LIN {X 0,Y 457.306,Z 988.134,A -85,B 0,C 180,E1 20807.433,E2 20807.433} C_VEL
LIN {X 0,Y 456.621,Z 997.32,A -85,B 0,C 180,E1 20804.572,E2 20804.572} C_VEL
LIN {X 0,Y 456.252,Z 1003.948,A -85,B 0,C 180,E1 20802.019,E2 20802.019} C_VEL
LIN {X 0,Y 456.036,Z 1009.804,A -85,B 0,C 180,E1 20799.213,E2 20799.213} C_VEL
LIN {X 0,Y 455.944,Z 1013.955,A -85,B 0,C 180,E1 20796.424,E2 20796.424} C_VEL
LIN {X 0,Y 455.898,Z 1016.711,A -85,B 0,C 180,E1 20793.65,E2 20793.65} C_VEL
LIN {X 0,Y 455.893,Z 1017.826,A -85,B 0,C 180,E1 20791.009,E2 20791.009} C_VEL
LIN {X 0,Y 455.907,Z 1017.736,A -85,B 0,C 180,E1 20788.495,E2 20788.495} C_VEL
LIN {X 0,Y 455.909,Z 1016.072,A -85,B 0,C 180,E1 20785.601,E2 20785.601} C_VEL
LIN {X 0,Y 455.929,Z 1013.324,A -85,B 0,C 180,E1 20783.076,E2 20783.076} C_VEL
LIN {X 0,Y 456.046,Z 1008.598,A -85,B 0,C 180,E1 20780.157,E2 20780.157} C_VEL
LIN {X 0,Y 456.297,Z 1003.054,A -85,B 0,C 180,E1 20777.603,E2 20777.603} C_VEL
LIN {X 0,Y 456.792,Z 994.97,A -85,B 0,C 180,E1 20774.646,E2 20774.646} C_VEL
LIN {X 0,Y 457.47,Z 986.327,A -85,B 0,C 180,E1 20772.055,E2 20772.055} C_VEL
LIN {X 0,Y 458.57,Z 974.884,A -85,B 0,C 180,E1 20769.186,E2 20769.186} C_VEL
LIN {X 0,Y 460.023,Z 962.425,A -85,B 0,C 180,E1 20766.521,E2 20766.521} C_VEL
LIN {X 0,Y 461.835,Z 948.135,A -85,B 0,C 180,E1 20763.933,E2 20763.933} C_VEL
LIN {X 0,Y 464.103,Z 931.673,A -85,B 0,C 180,E1 20761.362,E2 20761.362} C_VEL
LIN {X 0,Y 466.448,Z 915.582,A -85,B 0,C 180,E1 20759.187,E2 20759.187} C_VEL
LIN {X 0,Y 468.956,Z 897.768,A -85,B 0,C 180,E1 20757.144,E2 20757.144} C_VEL
LIN {X 0,Y 471.66,Z 878.612,A -85,B 0,C 180,E1 20755.238,E2 20755.238} C_VEL
LIN {X 0,Y 474.23,Z 859.23,A -85,B 0,C 180,E1 20753.599,E2 20753.599} C_VEL
LIN {X 0,Y 476.999,Z 837.541,A -85,B 0,C 180,E1 20752.038,E2 20752.038} C_VEL
LIN {X 0,Y 479.213,Z 818.309,A -85,B 0,C 180,E1 20750.878,E2 20750.878} C_VEL
LIN {X 0,Y 481.581,Z 794.779,A -85,B 0,C 180,E1 20749.71,E2 20749.71} C_VEL
LIN {X 0,Y 483.484,Z 773.134,A -85,B 0,C 180,E1 20748.864,E2 20748.864} C_VEL
LIN {X 0,Y 485.004,Z 750.7,A -85,B 0,C 180,E1 20748.207,E2 20748.207} C_VEL
LIN {X 0,Y 486.043,Z 728.316,A -85,B 0,C 180,E1 20747.734,E2 20747.734} C_VEL
LIN {X 0,Y 491.395,Z 520.554,A -85,B 0,C 180,E1 20744.158,E2 20744.158} C_VEL
LIN {X 0,Y 493.752,Z 431.767,A -85,B 0,C 180,E1 20742.581,E2 20742.581} C_VEL
LIN {X 0,Y 480.639,Z 411.465,A -85,B 0,C 180,E1 20740.421,E2 20740.421} C_VEL
LIN {X 0,Y 467.607,Z 392.801,A -85,B 0,C 180,E1 20738.088,E2 20738.088} C_VEL
LIN {X 0,Y 463.585,Z 387.256,A -85,B 0,C 180,E1 20737.305,E2 20737.305} C_VEL
LIN {X 0,Y 458.876,Z 378.323,A -85,B 0,C 180,E1 20735.575,E2 20735.575} C_VEL
LIN {X 0,Y 457.213,Z 375.183,A -85,B 0,C 180,E1 20734.917,E2 20734.917} C_VEL
LIN {X 0,Y 457.035,Z 374.27,A -85,B 0,C 180,E1 20734.665,E2 20734.665} C_VEL
LIN {X 0,Y 456.993,Z 374.085,A -85,B 0,C 180,E1 20731.087,E2 20731.087} C_VEL
LIN {X 0,Y 457.016,Z 374.122,A -85,B 0,C 180,E1 20727.492,E2 20727.492} C_VEL
LIN {X 0,Y 457.052,Z 374.11,A -85,B 0,C 180,E1 20723.873,E2 20723.873} C_VEL
LIN {X 0,Y 457.006,Z 374.114,A -85,B 0,C 180,E1 20720.356,E2 20720.356} C_VEL
LIN {X 0,Y 457,Z 374.117,A -85,B 0,C 180,E1 20716.655,E2 20716.655} C_VEL
LIN {X 0,Y 457.035,Z 374.118,A -85,B 0,C 180,E1 20713.151,E2 20713.151} C_VEL
LIN {X 0,Y 457.061,Z 374.117,A -85,B 0,C 180,E1 20709.443,E2 20709.443} C_VEL
LIN {X 0,Y 457.02,Z 374.12,A -85,B 0,C 180,E1 20705.901,E2 20705.901} C_VEL
LIN {X 0,Y 457.012,Z 374.117,A -85,B 0,C 180,E1 20702.257,E2 20702.257} C_VEL
LIN {X 0,Y 457.045,Z 374.111,A -85,B 0,C 180,E1 20698.746,E2 20698.746} C_VEL
LIN {X 0,Y 457.066,Z 374.108,A -85,B 0,C 180,E1 20695.105,E2 20695.105} C_VEL
LIN {X 0,Y 457.027,Z 374.117,A -85,B 0,C 180,E1 20691.571,E2 20691.571} C_VEL
LIN {X 0,Y 457.024,Z 374.114,A -85,B 0,C 180,E1 20687.876,E2 20687.876} C_VEL
LIN {X 0,Y 457.051,Z 374.108,A -85,B 0,C 180,E1 20684.252,E2 20684.252} C_VEL
LIN {X 0,Y 457.075,Z 374.104,A -85,B 0,C 180,E1 20680.579,E2 20680.579} C_VEL
LIN {X 0,Y 457.049,Z 374.11,A -85,B 0,C 180,E1 20676.946,E2 20676.946} C_VEL
LIN {X 0,Y 457.034,Z 374.112,A -85,B 0,C 180,E1 20673.353,E2 20673.353} C_VEL
LIN {X 0,Y 457.054,Z 374.105,A -85,B 0,C 180,E1 20669.771,E2 20669.771} C_VEL
LIN {X 0,Y 457.078,Z 374.103,A -85,B 0,C 180,E1 20666.095,E2 20666.095} C_VEL
LIN {X 0,Y 457.069,Z 374.106,A -85,B 0,C 180,E1 20662.355,E2 20662.355} C_VEL
LIN {X 0,Y 457.044,Z 374.106,A -85,B 0,C 180,E1 20658.805,E2 20658.805} C_VEL
LIN {X 0,Y 457.05,Z 374.113,A -85,B 0,C 180,E1 20655.04,E2 20655.04} C_VEL
LIN {X 0,Y 457.075,Z 374.112,A -85,B 0,C 180,E1 20651.342,E2 20651.342} C_VEL
LIN {X 0,Y 457.073,Z 374.105,A -85,B 0,C 180,E1 20647.607,E2 20647.607} C_VEL
LIN {X 0,Y 457.074,Z 374.108,A -85,B 0,C 180,E1 20643.9,E2 20643.9} C_VEL
LIN {X 0,Y 457.051,Z 374.08,A -85,B 0,C 180,E1 20640.204,E2 20640.204} C_VEL
LIN {X 0,Y 457.056,Z 374.087,A -85,B 0,C 180,E1 20636.5,E2 20636.5} C_VEL
LIN {X 0,Y 457.075,Z 374.098,A -85,B 0,C 180,E1 20632.775,E2 20632.775} C_VEL
LIN {X 0,Y 457.119,Z 374.398,A -85,B 0,C 180,E1 20631.555,E2 20631.555} C_VEL
LIN {X 0,Y 457.57,Z 376.045,A -85,B 0,C 180,E1 20631.29,E2 20631.29} C_VEL
LIN {X 0,Y 459.613,Z 379.002,A -85,B 0,C 180,E1 20630.876,E2 20630.876} C_VEL
LIN {X 0,Y 461.397,Z 380.643,A -85,B 0,C 180,E1 20630.548,E2 20630.548} C_VEL
LIN {X 0,Y 463.85,Z 384.388,A -85,B 0,C 180,E1 20630.067,E2 20630.067} C_VEL
LIN {X 0,Y 465.76,Z 386.443,A -85,B 0,C 180,E1 20629.721,E2 20629.721} C_VEL
LIN {X 0,Y 469.06,Z 390.773,A -85,B 0,C 180,E1 20629.118,E2 20629.118} C_VEL
LIN {X 0,Y 469.173,Z 390.881,A -85,B 0,C 180,E1 20629.098,E2 20629.098} C_VEL
LIN {X 0,Y 470.97,Z 393.832,A -85,B 0,C 180,E1 20628.762,E2 20628.762} C_VEL
LIN {X 0,Y 472.42,Z 399.823,A -85,B 0,C 180,E1 20628.407,E2 20628.407} C_VEL
LIN {X 0,Y 473.933,Z 407.518,A -85,B 0,C 180,E1 20628.004,E2 20628.004} C_VEL
LIN {X 0,Y 475.539,Z 410.916,A -85,B 0,C 180,E1 20627.694,E2 20627.694} C_VEL
LIN {X 0,Y 486.708,Z 426.723,A -85,B 0,C 180,E1 20625.82,E2 20625.82} C_VEL
LIN {X 0,Y 488.009,Z 429.058,A -85,B 0,C 180,E1 20625.601,E2 20625.601} C_VEL
LIN {X 0,Y 481.886,Z 639.66,A -85,B 0,C 180,E1 20621.903,E2 20621.903} C_VEL
LIN {X 0,Y 479.731,Z 713.742,A -85,B 0,C 180,E1 20620.595,E2 20620.595} C_VEL
LIN {X 0,Y 478.332,Z 735.919,A -85,B 0,C 180,E1 20620.01,E2 20620.01} C_VEL
LIN {X 0,Y 476.579,Z 758.024,A -85,B 0,C 180,E1 20619.232,E2 20619.232} C_VEL
LIN {X 0,Y 474.343,Z 779.679,A -85,B 0,C 180,E1 20618.237,E2 20618.237} C_VEL
LIN {X 0,Y 471.889,Z 800.765,A -85,B 0,C 180,E1 20617.056,E2 20617.056} C_VEL
LIN {X 0,Y 469.117,Z 821.678,A -85,B 0,C 180,E1 20615.623,E2 20615.623} C_VEL
LIN {X 0,Y 466.118,Z 842.401,A -85,B 0,C 180,E1 20613.933,E2 20613.933} C_VEL
LIN {X 0,Y 463.189,Z 861.498,A -85,B 0,C 180,E1 20612.1,E2 20612.1} C_VEL
LIN {X 0,Y 460.249,Z 880.136,A -85,B 0,C 180,E1 20609.997,E2 20609.997} C_VEL
LIN {X 0,Y 457.509,Z 897.277,A -85,B 0,C 180,E1 20607.742,E2 20607.742} C_VEL
LIN {X 0,Y 454.98,Z 913.876,A -85,B 0,C 180,E1 20605.207,E2 20605.207} C_VEL
LIN {X 0,Y 452.94,Z 928.382,A -85,B 0,C 180,E1 20602.641,E2 20602.641} C_VEL
LIN {X 0,Y 451.242,Z 941.581,A -85,B 0,C 180,E1 20599.916,E2 20599.916} C_VEL
LIN {X 0,Y 449.92,Z 953.436,A -85,B 0,C 180,E1 20597.026,E2 20597.026} C_VEL
LIN {X 0,Y 448.998,Z 963.452,A -85,B 0,C 180,E1 20594.1,E2 20594.1} C_VEL
LIN {X 0,Y 448.435,Z 971.383,A -85,B 0,C 180,E1 20591.269,E2 20591.269} C_VEL
LIN {X 0,Y 448.117,Z 977.788,A -85,B 0,C 180,E1 20588.395,E2 20588.395} C_VEL
LIN {X 0,Y 447.972,Z 982.717,A -85,B 0,C 180,E1 20585.469,E2 20585.469} C_VEL
LIN {X 0,Y 447.896,Z 985.964,A -85,B 0,C 180,E1 20582.619,E2 20582.619} C_VEL
LIN {X 0,Y 447.884,Z 987.645,A -85,B 0,C 180,E1 20579.846,E2 20579.846} C_VEL
LIN {X 0,Y 447.902,Z 987.873,A -85,B 0,C 180,E1 20577.072,E2 20577.072} C_VEL
LIN {X 0,Y 447.911,Z 986.601,A -85,B 0,C 180,E1 20574.127,E2 20574.127} C_VEL
LIN {X 0,Y 447.948,Z 983.891,A -85,B 0,C 180,E1 20571.316,E2 20571.316} C_VEL
LIN {X 0,Y 448.068,Z 979.465,A -85,B 0,C 180,E1 20568.379,E2 20568.379} C_VEL
LIN {X 0,Y 448.305,Z 973.564,A -85,B 0,C 180,E1 20565.537,E2 20565.537} C_VEL
LIN {X 0,Y 448.786,Z 966.02,A -85,B 0,C 180,E1 20562.672,E2 20562.672} C_VEL
LIN {X 0,Y 449.558,Z 956.85,A -85,B 0,C 180,E1 20559.832,E2 20559.832} C_VEL
LIN {X 0,Y 450.704,Z 945.891,A -85,B 0,C 180,E1 20556.997,E2 20556.997} C_VEL
LIN {X 0,Y 452.212,Z 933.708,A -85,B 0,C 180,E1 20554.32,E2 20554.32} C_VEL
LIN {X 0,Y 454.155,Z 919.628,A -85,B 0,C 180,E1 20551.673,E2 20551.673} C_VEL
LIN {X 0,Y 456.535,Z 903.606,A -85,B 0,C 180,E1 20549.088,E2 20549.088} C_VEL
LIN {X 0,Y 459.226,Z 886.698,A -85,B 0,C 180,E1 20546.726,E2 20546.726} C_VEL
LIN {X 0,Y 462.143,Z 868.394,A -85,B 0,C 180,E1 20544.545,E2 20544.545} C_VEL
LIN {X 0,Y 465.06,Z 849.746,A -85,B 0,C 180,E1 20542.634,E2 20542.634} C_VEL
LIN {X 0,Y 467.9,Z 830.401,A -85,B 0,C 180,E1 20540.957,E2 20540.957} C_VEL
LIN {X 0,Y 470.853,Z 808.986,A -85,B 0,C 180,E1 20539.388,E2 20539.388} C_VEL
LIN {X 0,Y 473.194,Z 790.015,A -85,B 0,C 180,E1 20538.224,E2 20538.224} C_VEL
LIN {X 0,Y 475.597,Z 767.361,A -85,B 0,C 180,E1 20537.083,E2 20537.083} C_VEL
LIN {X 0,Y 477.597,Z 745.324,A -85,B 0,C 180,E1 20536.206,E2 20536.206} C_VEL
LIN {X 0,Y 479.103,Z 723.137,A -85,B 0,C 180,E1 20535.552,E2 20535.552} C_VEL
LIN {X 0,Y 480.178,Z 699.844,A -85,B 0,C 180,E1 20535.06,E2 20535.06} C_VEL
LIN {X 0,Y 485.98,Z 497.309,A -85,B 0,C 180,E1 20531.514,E2 20531.514} C_VEL
LIN {X 0,Y 488.115,Z 428.611,A -85,B 0,C 180,E1 20530.266,E2 20530.266} C_VEL
LIN {X 0,Y 476.772,Z 412.129,A -85,B 0,C 180,E1 20528.29,E2 20528.29} C_VEL
LIN {X 0,Y 469.203,Z 401.84,A -85,B 0,C 180,E1 20526.854,E2 20526.854} C_VEL
LIN {X 0,Y 465.608,Z 397.083,A -85,B 0,C 180,E1 20526.132,E2 20526.132} C_VEL
LIN {X 0,Y 461.979,Z 392.324,A -85,B 0,C 180,E1 20525.38,E2 20525.38} C_VEL
LIN {X 0,Y 458.836,Z 388.242,A -85,B 0,C 180,E1 20524.688,E2 20524.688} C_VEL
LIN {X 0,Y 457.761,Z 386.899,A -85,B 0,C 180,E1 20524.448,E2 20524.448} C_VEL
LIN {X 0,Y 454.797,Z 383.552,A -85,B 0,C 180,E1 20523.782,E2 20523.782} C_VEL
LIN {X 0,Y 453.604,Z 381.346,A -85,B 0,C 180,E1 20523.482,E2 20523.482} C_VEL
LIN {X 0,Y 450.664,Z 378.906,A -85,B 0,C 180,E1 20522.798,E2 20522.798} C_VEL
LIN {X 0,Y 449.291,Z 375.976,A -85,B 0,C 180,E1 20522.366,E2 20522.366} C_VEL
LIN {X 0,Y 449.128,Z 375.128,A -85,B 0,C 180,E1 20521.914,E2 20521.914} C_VEL
LIN {X 0,Y 449.132,Z 375.098,A -85,B 0,C 180,E1 20518.214,E2 20518.214} C_VEL
LIN {X 0,Y 449.135,Z 375.095,A -85,B 0,C 180,E1 20514.507,E2 20514.507} C_VEL
LIN {X 0,Y 449.128,Z 375.103,A -85,B 0,C 180,E1 20510.777,E2 20510.777} C_VEL
LIN {X 0,Y 449.104,Z 375.107,A -85,B 0,C 180,E1 20507.137,E2 20507.137} C_VEL
LIN {X 0,Y 449.103,Z 375.106,A -85,B 0,C 180,E1 20503.443,E2 20503.443} C_VEL
LIN {X 0,Y 449.125,Z 375.104,A -85,B 0,C 180,E1 20499.815,E2 20499.815} C_VEL
LIN {X 0,Y 449.129,Z 375.095,A -85,B 0,C 180,E1 20496.206,E2 20496.206} C_VEL
LIN {X 0,Y 449.092,Z 375.106,A -85,B 0,C 180,E1 20492.558,E2 20492.558} C_VEL
LIN {X 0,Y 449.073,Z 375.108,A -85,B 0,C 180,E1 20488.9,E2 20488.9} C_VEL
LIN {X 0,Y 449.116,Z 375.414,A -85,B 0,C 180,E1 20487.022,E2 20487.022} C_VEL
LIN {X 0,Y 450.636,Z 378.913,A -85,B 0,C 180,E1 20486.158,E2 20486.158} C_VEL
LIN {X 0,Y 451.942,Z 380.731,A -85,B 0,C 180,E1 20485.657,E2 20485.657} C_VEL
LIN {X 0,Y 453.93,Z 384.473,A -85,B 0,C 180,E1 20484.831,E2 20484.831} C_VEL
LIN {X 0,Y 459.557,Z 392.132,A -85,B 0,C 180,E1 20483.523,E2 20483.523} C_VEL
LIN {X 0,Y 466.249,Z 401.457,A -85,B 0,C 180,E1 20482.101,E2 20482.101} C_VEL
LIN {X 0,Y 474.956,Z 414.182,A -85,B 0,C 180,E1 20480.396,E2 20480.396} C_VEL
LIN {X 0,Y 485.83,Z 431.636,A -85,B 0,C 180,E1 20478.436,E2 20478.436} C_VEL
LIN {X 0,Y 488.286,Z 435.985,A -85,B 0,C 180,E1 20478.011,E2 20478.011} C_VEL
LIN {X 0,Y 482.252,Z 637.01,A -85,B 0,C 180,E1 20474.448,E2 20474.448} C_VEL
LIN {X 0,Y 479.387,Z 739.278,A -85,B 0,C 180,E1 20472.658,E2 20472.658} C_VEL
LIN {X 0,Y 477.889,Z 762.53,A -85,B 0,C 180,E1 20472.062,E2 20472.062} C_VEL
LIN {X 0,Y 476.13,Z 784.668,A -85,B 0,C 180,E1 20471.296,E2 20471.296} C_VEL
LIN {X 0,Y 473.953,Z 806.141,A -85,B 0,C 180,E1 20470.328,E2 20470.328} C_VEL
LIN {X 0,Y 471.59,Z 827.058,A -85,B 0,C 180,E1 20469.187,E2 20469.187} C_VEL
LIN {X 0,Y 468.918,Z 847.716,A -85,B 0,C 180,E1 20467.811,E2 20467.811} C_VEL
LIN {X 0,Y 466.071,Z 868.762,A -85,B 0,C 180,E1 20466.156,E2 20466.156} C_VEL
LIN {X 0,Y 463.451,Z 886.719,A -85,B 0,C 180,E1 20464.5,E2 20464.5} C_VEL
LIN {X 0,Y 460.512,Z 906.579,A -85,B 0,C 180,E1 20462.373,E2 20462.373} C_VEL
LIN {X 0,Y 458.095,Z 922.885,A -85,B 0,C 180,E1 20460.353,E2 20460.353} C_VEL
LIN {X 0,Y 455.797,Z 938.318,A -85,B 0,C 180,E1 20458.135,E2 20458.135} C_VEL
LIN {X 0,Y 453.711,Z 952.715,A -85,B 0,C 180,E1 20455.733,E2 20455.733} C_VEL
LIN {X 0,Y 451.86,Z 966.427,A -85,B 0,C 180,E1 20453.06,E2 20453.06} C_VEL
LIN {X 0,Y 450.47,Z 978.243,A -85,B 0,C 180,E1 20450.397,E2 20450.397} C_VEL
LIN {X 0,Y 449.449,Z 988.133,A -85,B 0,C 180,E1 20447.747,E2 20447.747} C_VEL
LIN {X 0,Y 448.706,Z 997.277,A -85,B 0,C 180,E1 20444.851,E2 20444.851} C_VEL
LIN {X 0,Y 448.292,Z 1003.948,A -85,B 0,C 180,E1 20442.236,E2 20442.236} C_VEL
LIN {X 0,Y 448.044,Z 1009.804,A -85,B 0,C 180,E1 20439.379,E2 20439.379} C_VEL
LIN {X 0,Y 447.939,Z 1013.829,A -85,B 0,C 180,E1 20436.642,E2 20436.642} C_VEL
LIN {X 0,Y 447.904,Z 1016.678,A -85,B 0,C 180,E1 20433.775,E2 20433.775} C_VEL
LIN {X 0,Y 447.894,Z 1017.826,A -85,B 0,C 180,E1 20431.027,E2 20431.027} C_VEL
LIN {X 0,Y 447.907,Z 1017.736,A -85,B 0,C 180,E1 20428.468,E2 20428.468} C_VEL
LIN {X 0,Y 447.908,Z 1016.071,A -85,B 0,C 180,E1 20425.522,E2 20425.522} C_VEL
LIN {X 0,Y 447.93,Z 1013.324,A -85,B 0,C 180,E1 20422.952,E2 20422.952} C_VEL
LIN {X 0,Y 448.055,Z 1008.852,A -85,B 0,C 180,E1 20420.11,E2 20420.11} C_VEL
LIN {X 0,Y 448.338,Z 1003.053,A -85,B 0,C 180,E1 20417.38,E2 20417.38} C_VEL
LIN {X 0,Y 448.879,Z 994.969,A -85,B 0,C 180,E1 20414.368,E2 20414.368} C_VEL
LIN {X 0,Y 449.627,Z 986.287,A -85,B 0,C 180,E1 20411.72,E2 20411.72} C_VEL
LIN {X 0,Y 450.824,Z 974.882,A -85,B 0,C 180,E1 20408.812,E2 20408.812} C_VEL
LIN {X 0,Y 452.364,Z 962.645,A -85,B 0,C 180,E1 20406.146,E2 20406.146} C_VEL
LIN {X 0,Y 454.246,Z 948.903,A -85,B 0,C 180,E1 20403.605,E2 20403.605} C_VEL
LIN {X 0,Y 456.476,Z 933.887,A -85,B 0,C 180,E1 20401.181,E2 20401.181} C_VEL
LIN {X 0,Y 458.778,Z 918.343,A -85,B 0,C 180,E1 20399.052,E2 20399.052} C_VEL
LIN {X 0,Y 461.573,Z 899.832,A -85,B 0,C 180,E1 20396.846,E2 20396.846} C_VEL
LIN {X 0,Y 464.198,Z 882.341,A -85,B 0,C 180,E1 20395.049,E2 20395.049} C_VEL
LIN {X 0,Y 467.102,Z 862.087,A -85,B 0,C 180,E1 20393.258,E2 20393.258} C_VEL
LIN {X 0,Y 469.882,Z 842.001,A -85,B 0,C 180,E1 20391.747,E2 20391.747} C_VEL
LIN {X 0,Y 472.469,Z 821.129,A -85,B 0,C 180,E1 20390.438,E2 20390.438} C_VEL
LIN {X 0,Y 474.689,Z 801.401,A -85,B 0,C 180,E1 20389.399,E2 20389.399} C_VEL
LIN {X 0,Y 476.825,Z 778.64,A -85,B 0,C 180,E1 20388.442,E2 20388.442} C_VEL
LIN {X 0,Y 478.65,Z 755.746,A -85,B 0,C 180,E1 20387.702,E2 20387.702} C_VEL
LIN {X 0,Y 479.86,Z 733.001,A -85,B 0,C 180,E1 20387.192,E2 20387.192} C_VEL
LIN {X 0,Y 485.717,Z 522.344,A -85,B 0,C 180,E1 20383.518,E2 20383.518} C_VEL
LIN {X 0,Y 488.162,Z 435.454,A -85,B 0,C 180,E1 20381.956,E2 20381.956} C_VEL
LIN {X 0,Y 476.385,Z 417.117,A -85,B 0,C 180,E1 20379.959,E2 20379.959} C_VEL
LIN {X 0,Y 463.976,Z 399.188,A -85,B 0,C 180,E1 20377.696,E2 20377.696} C_VEL
LIN {X 0,Y 455.028,Z 386.977,A -85,B 0,C 180,E1 20375.922,E2 20375.922} C_VEL
LIN {X 0,Y 453.439,Z 383.957,A -85,B 0,C 180,E1 20375.335,E2 20375.335} C_VEL
LIN {X 0,Y 450.758,Z 379.036,A -85,B 0,C 180,E1 20374.292,E2 20374.292} C_VEL
LIN {X 0,Y 449.102,Z 375.342,A -85,B 0,C 180,E1 20373.46,E2 20373.46} C_VEL
LIN {X 0,Y 449.114,Z 375.057,A -85,B 0,C 180,E1 20370.01,E2 20370.01} C_VEL
LIN {X 0,Y 449.067,Z 375.102,A -85,B 0,C 180,E1 20366.442,E2 20366.442} C_VEL
LIN {X 0,Y 449.055,Z 375.101,A -85,B 0,C 180,E1 20362.794,E2 20362.794} C_VEL
LIN {X 0,Y 449.083,Z 375.107,A -85,B 0,C 180,E1 20359.239,E2 20359.239} C_VEL
LIN {X 0,Y 449.122,Z 375.105,A -85,B 0,C 180,E1 20355.627,E2 20355.627} C_VEL
LIN {X 0,Y 449.076,Z 375.108,A -85,B 0,C 180,E1 20352.08,E2 20352.08} C_VEL
LIN {X 0,Y 449.068,Z 375.104,A -85,B 0,C 180,E1 20348.45,E2 20348.45} C_VEL
LIN {X 0,Y 449.095,Z 375.096,A -85,B 0,C 180,E1 20344.853,E2 20344.853} C_VEL
LIN {X 0,Y 449.132,Z 375.093,A -85,B 0,C 180,E1 20341.148,E2 20341.148} C_VEL
LIN {X 0,Y 449.093,Z 375.097,A -85,B 0,C 180,E1 20337.575,E2 20337.575} C_VEL
LIN {X 0,Y 449.078,Z 375.096,A -85,B 0,C 180,E1 20333.993,E2 20333.993} C_VEL
LIN {X 0,Y 449.102,Z 375.097,A -85,B 0,C 180,E1 20330.388,E2 20330.388} C_VEL
LIN {X 0,Y 449.137,Z 375.093,A -85,B 0,C 180,E1 20326.744,E2 20326.744} C_VEL
LIN {X 0,Y 449.102,Z 375.096,A -85,B 0,C 180,E1 20323.176,E2 20323.176} C_VEL
LIN {X 0,Y 449.091,Z 375.096,A -85,B 0,C 180,E1 20319.54,E2 20319.54} C_VEL
LIN {X 0,Y 449.105,Z 375.098,A -85,B 0,C 180,E1 20315.882,E2 20315.882} C_VEL
LIN {X 0,Y 449.14,Z 375.095,A -85,B 0,C 180,E1 20312.272,E2 20312.272} C_VEL
LIN {X 0,Y 449.132,Z 375.096,A -85,B 0,C 180,E1 20308.49,E2 20308.49} C_VEL
LIN {X 0,Y 449.107,Z 375.101,A -85,B 0,C 180,E1 20304.783,E2 20304.783} C_VEL
LIN {X 0,Y 449.105,Z 375.104,A -85,B 0,C 180,E1 20301.11,E2 20301.11} C_VEL
LIN {X 0,Y 449.122,Z 375.102,A -85,B 0,C 180,E1 20297.407,E2 20297.407} C_VEL
LIN {X 0,Y 449.136,Z 375.093,A -85,B 0,C 180,E1 20293.633,E2 20293.633} C_VEL
LIN {X 0,Y 449.139,Z 375.094,A -85,B 0,C 180,E1 20289.871,E2 20289.871} C_VEL
LIN {X 0,Y 449.125,Z 375.102,A -85,B 0,C 180,E1 20286.086,E2 20286.086} C_VEL
LIN {X 0,Y 449.114,Z 375.097,A -85,B 0,C 180,E1 20282.443,E2 20282.443} C_VEL
LIN {X 0,Y 449.125,Z 375.091,A -85,B 0,C 180,E1 20278.7,E2 20278.7} C_VEL
LIN {X 0,Y 449.131,Z 375.069,A -85,B 0,C 180,E1 20275.018,E2 20275.018} C_VEL
LIN {X 0,Y 449.166,Z 375.317,A -85,B 0,C 180,E1 20272.922,E2 20272.922} C_VEL
LIN {X 0,Y 449.5,Z 376.685,A -85,B 0,C 180,E1 20272.649,E2 20272.649} C_VEL
LIN {X 0,Y 451.343,Z 379.691,A -85,B 0,C 180,E1 20272.239,E2 20272.239} C_VEL
LIN {X 0,Y 453.539,Z 381.571,A -85,B 0,C 180,E1 20271.812,E2 20271.812} C_VEL
LIN {X 0,Y 456.06,Z 385.452,A -85,B 0,C 180,E1 20271.288,E2 20271.288} C_VEL
LIN {X 0,Y 458.024,Z 387.57,A -85,B 0,C 180,E1 20270.911,E2 20270.911} C_VEL
LIN {X 0,Y 461.301,Z 391.883,A -85,B 0,C 180,E1 20270.276,E2 20270.276} C_VEL
LIN {X 0,Y 471.087,Z 404.835,A -85,B 0,C 180,E1 20268.477,E2 20268.477} C_VEL
LIN {X 0,Y 475.539,Z 410.916,A -85,B 0,C 180,E1 20267.694,E2 20267.694} C_VEL
LIN {X 0,Y 477.361,Z 414.858,A -85,B 0,C 180,E1 20267.346,E2 20267.346} C_VEL
LIN {X 0,Y 480.094,Z 427.929,A -85,B 0,C 180,E1 20266.67,E2 20266.67} C_VEL
LIN {X 0,Y 481.704,Z 431.334,A -85,B 0,C 180,E1 20266.376,E2 20266.376} C_VEL
LIN {X 0,Y 482.501,Z 432.851,A -85,B 0,C 180,E1 20266.236,E2 20266.236} C_VEL
LIN {X 0,Y 476.005,Z 642.981,A -85,B 0,C 180,E1 20262.511,E2 20262.511} C_VEL
LIN {X 0,Y 473.803,Z 714.075,A -85,B 0,C 180,E1 20261.241,E2 20261.241} C_VEL
LIN {X 0,Y 472.324,Z 736.363,A -85,B 0,C 180,E1 20260.648,E2 20260.648} C_VEL
LIN {X 0,Y 470.516,Z 758.088,A -85,B 0,C 180,E1 20259.877,E2 20259.877} C_VEL
LIN {X 0,Y 468.233,Z 779.223,A -85,B 0,C 180,E1 20258.903,E2 20258.903} C_VEL
LIN {X 0,Y 465.639,Z 800.479,A -85,B 0,C 180,E1 20257.709,E2 20257.709} C_VEL
LIN {X 0,Y 462.793,Z 820.681,A -85,B 0,C 180,E1 20256.322,E2 20256.322} C_VEL
LIN {X 0,Y 459.634,Z 841.642,A -85,B 0,C 180,E1 20254.613,E2 20254.613} C_VEL
LIN {X 0,Y 456.61,Z 860.307,A -85,B 0,C 180,E1 20252.821,E2 20252.821} C_VEL
LIN {X 0,Y 453.443,Z 879.153,A -85,B 0,C 180,E1 20250.692,E2 20250.692} C_VEL
LIN {X 0,Y 450.582,Z 896.071,A -85,B 0,C 180,E1 20248.471,E2 20248.471} C_VEL
LIN {X 0,Y 447.814,Z 912.788,A -85,B 0,C 180,E1 20245.9,E2 20245.9} C_VEL
LIN {X 0,Y 445.339,Z 928.656,A -85,B 0,C 180,E1 20243.033,E2 20243.033} C_VEL
LIN {X 0,Y 443.511,Z 941.818,A -85,B 0,C 180,E1 20240.263,E2 20240.263} C_VEL
LIN {X 0,Y 442.086,Z 953.636,A -85,B 0,C 180,E1 20237.324,E2 20237.324} C_VEL
LIN {X 0,Y 441.097,Z 963.606,A -85,B 0,C 180,E1 20234.348,E2 20234.348} C_VEL
LIN {X 0,Y 440.461,Z 971.85,A -85,B 0,C 180,E1 20231.33,E2 20231.33} C_VEL
LIN {X 0,Y 440.124,Z 978.144,A -85,B 0,C 180,E1 20228.403,E2 20228.403} C_VEL
LIN {X 0,Y 439.97,Z 983.026,A -85,B 0,C 180,E1 20225.372,E2 20225.372} C_VEL
LIN {X 0,Y 439.894,Z 986.215,A -85,B 0,C 180,E1 20222.372,E2 20222.372} C_VEL
LIN {X 0,Y 439.892,Z 987.764,A -85,B 0,C 180,E1 20219.542,E2 20219.542} C_VEL
LIN {X 0,Y 439.906,Z 987.83,A -85,B 0,C 180,E1 20216.765,E2 20216.765} C_VEL
LIN {X 0,Y 439.903,Z 986.508,A -85,B 0,C 180,E1 20213.934,E2 20213.934} C_VEL
LIN {X 0,Y 439.951,Z 983.616,A -85,B 0,C 180,E1 20210.982,E2 20210.982} C_VEL
LIN {X 0,Y 440.085,Z 979.061,A -85,B 0,C 180,E1 20207.982,E2 20207.982} C_VEL
LIN {X 0,Y 440.373,Z 973.045,A -85,B 0,C 180,E1 20205.077,E2 20205.077} C_VEL
LIN {X 0,Y 440.936,Z 965.297,A -85,B 0,C 180,E1 20202.138,E2 20202.138} C_VEL
LIN {X 0,Y 441.803,Z 956.093,A -85,B 0,C 180,E1 20199.284,E2 20199.284} C_VEL
LIN {X 0,Y 443.125,Z 944.721,A -85,B 0,C 180,E1 20196.336,E2 20196.336} C_VEL
LIN {X 0,Y 444.942,Z 931.293,A -85,B 0,C 180,E1 20193.406,E2 20193.406} C_VEL
LIN {X 0,Y 447.185,Z 916.519,A -85,B 0,C 180,E1 20190.65,E2 20190.65} C_VEL
LIN {X 0,Y 449.8,Z 900.719,A -85,B 0,C 180,E1 20188.116,E2 20188.116} C_VEL
LIN {X 0,Y 452.68,Z 883.881,A -85,B 0,C 180,E1 20185.794,E2 20185.794} C_VEL
LIN {X 0,Y 455.585,Z 866.7,A -85,B 0,C 180,E1 20183.765,E2 20183.765} C_VEL
LIN {X 0,Y 458.855,Z 846.667,A -85,B 0,C 180,E1 20181.743,E2 20181.743} C_VEL
LIN {X 0,Y 461.8,Z 827.975,A -85,B 0,C 180,E1 20180.137,E2 20180.137} C_VEL
LIN {X 0,Y 464.603,Z 808.205,A -85,B 0,C 180,E1 20178.703,E2 20178.703} C_VEL
LIN {X 0,Y 467.301,Z 787.401,A -85,B 0,C 180,E1 20177.431,E2 20177.431} C_VEL
LIN {X 0,Y 469.61,Z 766.215,A -85,B 0,C 180,E1 20176.386,E2 20176.386} C_VEL
LIN {X 0,Y 471.744,Z 743.666,A -85,B 0,C 180,E1 20175.501,E2 20175.501} C_VEL
LIN {X 0,Y 473.209,Z 722.444,A -85,B 0,C 180,E1 20174.884,E2 20174.884} C_VEL
LIN {X 0,Y 474.333,Z 697.976,A -85,B 0,C 180,E1 20174.374,E2 20174.374} C_VEL
LIN {X 0,Y 480.528,Z 497.169,A -85,B 0,C 180,E1 20170.813,E2 20170.813} C_VEL
LIN {X 0,Y 482.667,Z 432.394,A -85,B 0,C 180,E1 20169.619,E2 20169.619} C_VEL
LIN {X 0,Y 470.299,Z 414.39,A -85,B 0,C 180,E1 20167.36,E2 20167.36} C_VEL
LIN {X 0,Y 461.96,Z 403.303,A -85,B 0,C 180,E1 20165.683,E2 20165.683} C_VEL
LIN {X 0,Y 458.411,Z 398.642,A -85,B 0,C 180,E1 20164.915,E2 20164.915} C_VEL
LIN {X 0,Y 454.674,Z 393.744,A -85,B 0,C 180,E1 20164.067,E2 20164.067} C_VEL
LIN {X 0,Y 451.48,Z 389.865,A -85,B 0,C 180,E1 20163.324,E2 20163.324} C_VEL
LIN {X 0,Y 450.425,Z 388.275,A -85,B 0,C 180,E1 20163.054,E2 20163.054} C_VEL
LIN {X 0,Y 447.385,Z 385.155,A -85,B 0,C 180,E1 20162.306,E2 20162.306} C_VEL
LIN {X 0,Y 445.791,Z 382.391,A -85,B 0,C 180,E1 20161.864,E2 20161.864} C_VEL
LIN {X 0,Y 442.79,Z 379.979,A -85,B 0,C 180,E1 20161.1,E2 20161.1} C_VEL
LIN {X 0,Y 441.345,Z 376.941,A -85,B 0,C 180,E1 20160.585,E2 20160.585} C_VEL
LIN {X 0,Y 441.206,Z 376.121,A -85,B 0,C 180,E1 20160.13,E2 20160.13} C_VEL
LIN {X 0,Y 441.194,Z 376.092,A -85,B 0,C 180,E1 20156.232,E2 20156.232} C_VEL
LIN {X 0,Y 441.199,Z 376.081,A -85,B 0,C 180,E1 20152.448,E2 20152.448} C_VEL
LIN {X 0,Y 441.192,Z 376.091,A -85,B 0,C 180,E1 20148.629,E2 20148.629} C_VEL
LIN {X 0,Y 441.168,Z 376.092,A -85,B 0,C 180,E1 20144.893,E2 20144.893} C_VEL
LIN {X 0,Y 441.157,Z 376.096,A -85,B 0,C 180,E1 20141.227,E2 20141.227} C_VEL
LIN {X 0,Y 441.161,Z 376.097,A -85,B 0,C 180,E1 20137.479,E2 20137.479} C_VEL
LIN {X 0,Y 441.186,Z 376.092,A -85,B 0,C 180,E1 20133.774,E2 20133.774} C_VEL
LIN {X 0,Y 441.179,Z 376.083,A -85,B 0,C 180,E1 20130.094,E2 20130.094} C_VEL
LIN {X 0,Y 441.184,Z 376.422,A -85,B 0,C 180,E1 20128.668,E2 20128.668} C_VEL
LIN {X 0,Y 442.902,Z 380.137,A -85,B 0,C 180,E1 20127.655,E2 20127.655} C_VEL
LIN {X 0,Y 444.155,Z 381.939,A -85,B 0,C 180,E1 20127.109,E2 20127.109} C_VEL
LIN {X 0,Y 446.08,Z 385.187,A -85,B 0,C 180,E1 20126.422,E2 20126.422} C_VEL
LIN {X 0,Y 448.236,Z 387.81,A -85,B 0,C 180,E1 20125.875,E2 20125.875} C_VEL
LIN {X 0,Y 452.636,Z 393.643,A -85,B 0,C 180,E1 20124.793,E2 20124.793} C_VEL
LIN {X 0,Y 456.797,Z 399.453,A -85,B 0,C 180,E1 20123.812,E2 20123.812} C_VEL
LIN {X 0,Y 462.878,Z 408.014,A -85,B 0,C 180,E1 20122.492,E2 20122.492} C_VEL
LIN {X 0,Y 471.783,Z 421.318,A -85,B 0,C 180,E1 20120.698,E2 20120.698} C_VEL
LIN {X 0,Y 482.373,Z 438.559,A -85,B 0,C 180,E1 20118.746,E2 20118.746} C_VEL
LIN {X 0,Y 482.844,Z 439.75,A -85,B 0,C 180,E1 20118.654,E2 20118.654} C_VEL
LIN {X 0,Y 476.417,Z 638.988,A -85,B 0,C 180,E1 20115.079,E2 20115.079} C_VEL
LIN {X 0,Y 473.404,Z 739.112,A -85,B 0,C 180,E1 20113.303,E2 20113.303} C_VEL
LIN {X 0,Y 471.806,Z 762.399,A -85,B 0,C 180,E1 20112.702,E2 20112.702} C_VEL
LIN {X 0,Y 469.93,Z 784.664,A -85,B 0,C 180,E1 20111.922,E2 20111.922} C_VEL
LIN {X 0,Y 467.711,Z 805.413,A -85,B 0,C 180,E1 20110.98,E2 20110.98} C_VEL
LIN {X 0,Y 465.218,Z 826.393,A -85,B 0,C 180,E1 20109.829,E2 20109.829} C_VEL
LIN {X 0,Y 462.375,Z 847.095,A -85,B 0,C 180,E1 20108.443,E2 20108.443} C_VEL
LIN {X 0,Y 459.463,Z 867.441,A -85,B 0,C 180,E1 20106.839,E2 20106.839} C_VEL
LIN {X 0,Y 456.673,Z 885.522,A -85,B 0,C 180,E1 20105.16,E2 20105.16} C_VEL
LIN {X 0,Y 453.67,Z 904.543,A -85,B 0,C 180,E1 20103.124,E2 20103.124} C_VEL
LIN {X 0,Y 451.086,Z 920.836,A -85,B 0,C 180,E1 20101.098,E2 20101.098} C_VEL
LIN {X 0,Y 448.404,Z 937.944,A -85,B 0,C 180,E1 20098.65,E2 20098.65} C_VEL
LIN {X 0,Y 446.356,Z 951.783,A -85,B 0,C 180,E1 20096.362,E2 20096.362} C_VEL
LIN {X 0,Y 444.306,Z 965.79,A -85,B 0,C 180,E1 20093.616,E2 20093.616} C_VEL
LIN {X 0,Y 442.77,Z 977.711,A -85,B 0,C 180,E1 20090.906,E2 20090.906} C_VEL
LIN {X 0,Y 441.599,Z 988.132,A -85,B 0,C 180,E1 20088.074,E2 20088.074} C_VEL
LIN {X 0,Y 440.792,Z 997.277,A -85,B 0,C 180,E1 20085.124,E2 20085.124} C_VEL
LIN {X 0,Y 440.314,Z 1004.25,A -85,B 0,C 180,E1 20082.328,E2 20082.328} C_VEL
LIN {X 0,Y 440.046,Z 1010.218,A -85,B 0,C 180,E1 20079.287,E2 20079.287} C_VEL
LIN {X 0,Y 439.939,Z 1013.955,A -85,B 0,C 180,E1 20076.659,E2 20076.659} C_VEL
LIN {X 0,Y 439.905,Z 1016.711,A -85,B 0,C 180,E1 20073.783,E2 20073.783} C_VEL
LIN {X 0,Y 439.895,Z 1017.825,A -85,B 0,C 180,E1 20071.045,E2 20071.045} C_VEL
LIN {X 0,Y 439.907,Z 1017.736,A -85,B 0,C 180,E1 20068.441,E2 20068.441} C_VEL
LIN {X 0,Y 439.907,Z 1016.071,A -85,B 0,C 180,E1 20065.441,E2 20065.441} C_VEL
LIN {X 0,Y 439.933,Z 1013.324,A -85,B 0,C 180,E1 20062.823,E2 20062.823} C_VEL
LIN {X 0,Y 440.086,Z 1008.597,A -85,B 0,C 180,E1 20059.796,E2 20059.796} C_VEL
LIN {X 0,Y 440.385,Z 1003.053,A -85,B 0,C 180,E1 20057.148,E2 20057.148} C_VEL
LIN {X 0,Y 440.987,Z 994.77,A -85,B 0,C 180,E1 20054.015,E2 20054.015} C_VEL
LIN {X 0,Y 441.842,Z 985.866,A -85,B 0,C 180,E1 20051.261,E2 20051.261} C_VEL
LIN {X 0,Y 443.129,Z 974.671,A -85,B 0,C 180,E1 20048.374,E2 20048.374} C_VEL
LIN {X 0,Y 444.761,Z 962.647,A -85,B 0,C 180,E1 20045.712,E2 20045.712} C_VEL
LIN {X 0,Y 446.667,Z 949.644,A -85,B 0,C 180,E1 20043.265,E2 20043.265} C_VEL
LIN {X 0,Y 449.001,Z 934.464,A -85,B 0,C 180,E1 20040.8,E2 20040.8} C_VEL
LIN {X 0,Y 451.636,Z 917.675,A -85,B 0,C 180,E1 20038.466,E2 20038.466} C_VEL
LIN {X 0,Y 454.686,Z 898.811,A -85,B 0,C 180,E1 20036.202,E2 20036.202} C_VEL
LIN {X 0,Y 457.454,Z 881.404,A -85,B 0,C 180,E1 20034.397,E2 20034.397} C_VEL
LIN {X 0,Y 460.5,Z 861.447,A -85,B 0,C 180,E1 20032.624,E2 20032.624} C_VEL
LIN {X 0,Y 463.421,Z 841.547,A -85,B 0,C 180,E1 20031.114,E2 20031.114} C_VEL
LIN {X 0,Y 466.183,Z 820.344,A -85,B 0,C 180,E1 20029.777,E2 20029.777} C_VEL
LIN {X 0,Y 468.666,Z 799.401,A -85,B 0,C 180,E1 20028.673,E2 20028.673} C_VEL
LIN {X 0,Y 470.88,Z 776.81,A -85,B 0,C 180,E1 20027.74,E2 20027.74} C_VEL
LIN {X 0,Y 472.785,Z 753.461,A -85,B 0,C 180,E1 20027.004,E2 20027.004} C_VEL
LIN {X 0,Y 473.979,Z 731.58,A -85,B 0,C 180,E1 20026.516,E2 20026.516} C_VEL
LIN {X 0,Y 480.209,Z 520.539,A -85,B 0,C 180,E1 20022.799,E2 20022.799} C_VEL
LIN {X 0,Y 482.667,Z 439.247,A -85,B 0,C 180,E1 20021.322,E2 20021.322} C_VEL
LIN {X 0,Y 472.135,Z 422.7,A -85,B 0,C 180,E1 20019.483,E2 20019.483} C_VEL
LIN {X 0,Y 460.227,Z 405.407,A -85,B 0,C 180,E1 20017.271,E2 20017.271} C_VEL
LIN {X 0,Y 449.057,Z 390.216,A -85,B 0,C 180,E1 20015.022,E2 20015.022} C_VEL
LIN {X 0,Y 446.352,Z 386.118,A -85,B 0,C 180,E1 20014.367,E2 20014.367} C_VEL
LIN {X 0,Y 443.106,Z 380.462,A -85,B 0,C 180,E1 20013.097,E2 20013.097} C_VEL
LIN {X 0,Y 441.338,Z 377.053,A -85,B 0,C 180,E1 20012.32,E2 20012.32} C_VEL
LIN {X 0,Y 441.188,Z 376.188,A -85,B 0,C 180,E1 20012.026,E2 20012.026} C_VEL
LIN {X 0,Y 441.132,Z 376.075,A -85,B 0,C 180,E1 20008.423,E2 20008.423} C_VEL
LIN {X 0,Y 441.117,Z 376.101,A -85,B 0,C 180,E1 20004.792,E2 20004.792} C_VEL
LIN {X 0,Y 441.13,Z 376.097,A -85,B 0,C 180,E1 20001.123,E2 20001.123} C_VEL
LIN {X 0,Y 441.167,Z 376.086,A -85,B 0,C 180,E1 19997.435,E2 19997.435} C_VEL
LIN {X 0,Y 441.164,Z 376.086,A -85,B 0,C 180,E1 19993.766,E2 19993.766} C_VEL
LIN {X 0,Y 441.133,Z 376.094,A -85,B 0,C 180,E1 19990.183,E2 19990.183} C_VEL
LIN {X 0,Y 441.131,Z 376.097,A -85,B 0,C 180,E1 19986.376,E2 19986.376} C_VEL
LIN {X 0,Y 441.153,Z 376.095,A -85,B 0,C 180,E1 19982.728,E2 19982.728} C_VEL
LIN {X 0,Y 441.195,Z 376.09,A -85,B 0,C 180,E1 19979.091,E2 19979.091} C_VEL
LIN {X 0,Y 441.17,Z 376.091,A -85,B 0,C 180,E1 19975.32,E2 19975.32} C_VEL
LIN {X 0,Y 441.144,Z 376.096,A -85,B 0,C 180,E1 19971.79,E2 19971.79} C_VEL
LIN {X 0,Y 441.149,Z 376.092,A -85,B 0,C 180,E1 19967.964,E2 19967.964} C_VEL
LIN {X 0,Y 441.18,Z 376.085,A -85,B 0,C 180,E1 19964.354,E2 19964.354} C_VEL
LIN {X 0,Y 441.195,Z 376.083,A -85,B 0,C 180,E1 19960.678,E2 19960.678} C_VEL
LIN {X 0,Y 441.172,Z 376.087,A -85,B 0,C 180,E1 19956.934,E2 19956.934} C_VEL
LIN {X 0,Y 441.157,Z 376.087,A -85,B 0,C 180,E1 19953.238,E2 19953.238} C_VEL
LIN {X 0,Y 441.161,Z 376.083,A -85,B 0,C 180,E1 19949.446,E2 19949.446} C_VEL
LIN {X 0,Y 441.186,Z 376.082,A -85,B 0,C 180,E1 19945.802,E2 19945.802} C_VEL
LIN {X 0,Y 441.201,Z 376.083,A -85,B 0,C 180,E1 19942.051,E2 19942.051} C_VEL
LIN {X 0,Y 441.196,Z 376.087,A -85,B 0,C 180,E1 19938.219,E2 19938.219} C_VEL
LIN {X 0,Y 441.178,Z 376.095,A -85,B 0,C 180,E1 19934.444,E2 19934.444} C_VEL
LIN {X 0,Y 441.171,Z 376.09,A -85,B 0,C 180,E1 19930.74,E2 19930.74} C_VEL
LIN {X 0,Y 441.186,Z 376.082,A -85,B 0,C 180,E1 19927.067,E2 19927.067} C_VEL
LIN {X 0,Y 441.197,Z 376.092,A -85,B 0,C 180,E1 19923.254,E2 19923.254} C_VEL
LIN {X 0,Y 441.194,Z 376.059,A -85,B 0,C 180,E1 19919.452,E2 19919.452} C_VEL
LIN {X 0,Y 441.191,Z 376.053,A -85,B 0,C 180,E1 19915.644,E2 19915.644} C_VEL
LIN {X 0,Y 441.211,Z 376.293,A -85,B 0,C 180,E1 19914.354,E2 19914.354} C_VEL
LIN {X 0,Y 441.619,Z 377.871,A -85,B 0,C 180,E1 19914.033,E2 19914.033} C_VEL
LIN {X 0,Y 443.524,Z 380.803,A -85,B 0,C 180,E1 19913.595,E2 19913.595} C_VEL
LIN {X 0,Y 445.716,Z 382.608,A -85,B 0,C 180,E1 19913.152,E2 19913.152} C_VEL
LIN {X 0,Y 448.145,Z 386.421,A -85,B 0,C 180,E1 19912.613,E2 19912.613} C_VEL
LIN {X 0,Y 450.321,Z 388.651,A -85,B 0,C 180,E1 19912.172,E2 19912.172} C_VEL
LIN {X 0,Y 453.532,Z 392.912,A -85,B 0,C 180,E1 19911.511,E2 19911.511} C_VEL
LIN {X 0,Y 463.582,Z 406.088,A -85,B 0,C 180,E1 19909.565,E2 19909.565} C_VEL
LIN {X 0,Y 474.527,Z 421.016,A -85,B 0,C 180,E1 19907.601,E2 19907.601} C_VEL
LIN {X 0,Y 481.704,Z 431.334,A -85,B 0,C 180,E1 19906.376,E2 19906.376} C_VEL
LIN {X 0,Y 482.678,Z 433.734,A -85,B 0,C 180,E1 19906.193,E2 19906.193} C_VEL
LIN {X 0,Y 482.97,Z 437.692,A -85,B 0,C 180,E1 19906.067,E2 19906.067} C_VEL
LIN {X 0,Y 481.945,Z 444.176,A -85,B 0,C 180,E1 19906.058,E2 19906.058} C_VEL
LIN {X 0,Y 476.888,Z 460.428,A -85,B 0,C 180,E1 19906.368,E2 19906.368} C_VEL
LIN {X 0,Y 476.02,Z 466.557,A -85,B 0,C 180,E1 19906.345,E2 19906.345} C_VEL
LIN {X 0,Y 469.317,Z 674.935,A -85,B 0,C 180,E1 19902.627,E2 19902.627} C_VEL
LIN {X 0,Y 467.827,Z 716.25,A -85,B 0,C 180,E1 19901.859,E2 19901.859} C_VEL
LIN {X 0,Y 466.314,Z 737.604,A -85,B 0,C 180,E1 19901.275,E2 19901.275} C_VEL
LIN {X 0,Y 464.36,Z 759.543,A -85,B 0,C 180,E1 19900.479,E2 19900.479} C_VEL
LIN {X 0,Y 462.046,Z 779.936,A -85,B 0,C 180,E1 19899.525,E2 19899.525} C_VEL
LIN {X 0,Y 459.316,Z 801.127,A -85,B 0,C 180,E1 19898.32,E2 19898.32} C_VEL
LIN {X 0,Y 456.314,Z 821.323,A -85,B 0,C 180,E1 19896.918,E2 19896.918} C_VEL
LIN {X 0,Y 452.979,Z 842.24,A -85,B 0,C 180,E1 19895.189,E2 19895.189} C_VEL
LIN {X 0,Y 449.999,Z 859.651,A -85,B 0,C 180,E1 19893.5,E2 19893.5} C_VEL
LIN {X 0,Y 446.603,Z 878.678,A -85,B 0,C 180,E1 19891.344,E2 19891.344} C_VEL
LIN {X 0,Y 443.57,Z 895.713,A -85,B 0,C 180,E1 19889.093,E2 19889.093} C_VEL
LIN {X 0,Y 440.703,Z 911.71,A -85,B 0,C 180,E1 19886.615,E2 19886.615} C_VEL
LIN {X 0,Y 438.104,Z 927.076,A -85,B 0,C 180,E1 19883.839,E2 19883.839} C_VEL
LIN {X 0,Y 435.957,Z 940.883,A -85,B 0,C 180,E1 19880.892,E2 19880.892} C_VEL
LIN {X 0,Y 434.424,Z 952.425,A -85,B 0,C 180,E1 19878.008,E2 19878.008} C_VEL
LIN {X 0,Y 433.319,Z 962.469,A -85,B 0,C 180,E1 19875.02,E2 19875.02} C_VEL
LIN {X 0,Y 432.618,Z 970.562,A -85,B 0,C 180,E1 19872.095,E2 19872.095} C_VEL
LIN {X 0,Y 432.176,Z 977.416,A -85,B 0,C 180,E1 19868.983,E2 19868.983} C_VEL
LIN {X 0,Y 431.984,Z 982.254,A -85,B 0,C 180,E1 19866.101,E2 19866.101} C_VEL
LIN {X 0,Y 431.914,Z 985.649,A -85,B 0,C 180,E1 19863.163,E2 19863.163} C_VEL
LIN {X 0,Y 431.896,Z 987.5,A -85,B 0,C 180,E1 19860.244,E2 19860.244} C_VEL
LIN {X 0,Y 431.897,Z 987.918,A -85,B 0,C 180,E1 19857.354,E2 19857.354} C_VEL
LIN {X 0,Y 431.913,Z 986.948,A -85,B 0,C 180,E1 19854.473,E2 19854.473} C_VEL
LIN {X 0,Y 431.943,Z 984.371,A -85,B 0,C 180,E1 19851.481,E2 19851.481} C_VEL
LIN {X 0,Y 432.065,Z 980.317,A -85,B 0,C 180,E1 19848.557,E2 19848.557} C_VEL
LIN {X 0,Y 432.342,Z 974.328,A -85,B 0,C 180,E1 19845.423,E2 19845.423} C_VEL
LIN {X 0,Y 432.91,Z 966.7,A -85,B 0,C 180,E1 19842.344,E2 19842.344} C_VEL
LIN {X 0,Y 433.783,Z 957.86,A -85,B 0,C 180,E1 19839.448,E2 19839.448} C_VEL
LIN {X 0,Y 435.084,Z 947.175,A -85,B 0,C 180,E1 19836.528,E2 19836.528} C_VEL
LIN {X 0,Y 437.011,Z 933.88,A -85,B 0,C 180,E1 19833.463,E2 19833.463} C_VEL
LIN {X 0,Y 439.297,Z 920.01,A -85,B 0,C 180,E1 19830.729,E2 19830.729} C_VEL
LIN {X 0,Y 442.048,Z 904.358,A -85,B 0,C 180,E1 19828.096,E2 19828.096} C_VEL
LIN {X 0,Y 444.824,Z 888.82,A -85,B 0,C 180,E1 19825.854,E2 19825.854} C_VEL
LIN {X 0,Y 448.094,Z 870.754,A -85,B 0,C 180,E1 19823.612,E2 19823.612} C_VEL
LIN {X 0,Y 451.126,Z 853.527,A -85,B 0,C 180,E1 19821.77,E2 19821.77} C_VEL
LIN {X 0,Y 454.354,Z 834.108,A -85,B 0,C 180,E1 19820.001,E2 19820.001} C_VEL
LIN {X 0,Y 457.493,Z 814.26,A -85,B 0,C 180,E1 19818.461,E2 19818.461} C_VEL
LIN {X 0,Y 460.229,Z 794.452,A -85,B 0,C 180,E1 19817.186,E2 19817.186} C_VEL
LIN {X 0,Y 462.766,Z 774.142,A -85,B 0,C 180,E1 19816.088,E2 19816.088} C_VEL
LIN {X 0,Y 465.024,Z 751.778,A -85,B 0,C 180,E1 19815.129,E2 19815.129} C_VEL
LIN {X 0,Y 466.93,Z 728.843,A -85,B 0,C 180,E1 19814.375,E2 19814.375} C_VEL
LIN {X 0,Y 468.188,Z 706.504,A -85,B 0,C 180,E1 19813.863,E2 19813.863} C_VEL
LIN {X 0,Y 475.143,Z 498.005,A -85,B 0,C 180,E1 19810.111,E2 19810.111} C_VEL
LIN {X 0,Y 477.327,Z 436.436,A -85,B 0,C 180,E1 19808.963,E2 19808.963} C_VEL
LIN {X 0,Y 466.443,Z 420.386,A -85,B 0,C 180,E1 19806.895,E2 19806.895} C_VEL
LIN {X 0,Y 458.378,Z 409.505,A -85,B 0,C 180,E1 19805.226,E2 19805.226} C_VEL
LIN {X 0,Y 455.027,Z 405.07,A -85,B 0,C 180,E1 19804.474,E2 19804.474} C_VEL
LIN {X 0,Y 451.336,Z 400.286,A -85,B 0,C 180,E1 19803.62,E2 19803.62} C_VEL
LIN {X 0,Y 447.974,Z 395.706,A -85,B 0,C 180,E1 19802.783,E2 19802.783} C_VEL
LIN {X 0,Y 444.351,Z 391.709,A -85,B 0,C 180,E1 19801.864,E2 19801.864} C_VEL
LIN {X 0,Y 443,Z 389.567,A -85,B 0,C 180,E1 19801.488,E2 19801.488} C_VEL
LIN {X 0,Y 439.928,Z 386.624,A -85,B 0,C 180,E1 19800.652,E2 19800.652} C_VEL
LIN {X 0,Y 438.303,Z 383.608,A -85,B 0,C 180,E1 19800.131,E2 19800.131} C_VEL
LIN {X 0,Y 435.099,Z 381.278,A -85,B 0,C 180,E1 19799.21,E2 19799.21} C_VEL
LIN {X 0,Y 433.416,Z 377.961,A -85,B 0,C 180,E1 19798.546,E2 19798.546} C_VEL
LIN {X 0,Y 433.255,Z 377.113,A -85,B 0,C 180,E1 19798.017,E2 19798.017} C_VEL
LIN {X 0,Y 433.259,Z 377.076,A -85,B 0,C 180,E1 19794.172,E2 19794.172} C_VEL
LIN {X 0,Y 433.258,Z 377.079,A -85,B 0,C 180,E1 19790.302,E2 19790.302} C_VEL
LIN {X 0,Y 433.256,Z 377.08,A -85,B 0,C 180,E1 19786.522,E2 19786.522} C_VEL
LIN {X 0,Y 433.229,Z 377.085,A -85,B 0,C 180,E1 19782.818,E2 19782.818} C_VEL
LIN {X 0,Y 433.215,Z 377.085,A -85,B 0,C 180,E1 19779.039,E2 19779.039} C_VEL
LIN {X 0,Y 433.214,Z 377.08,A -85,B 0,C 180,E1 19775.308,E2 19775.308} C_VEL
LIN {X 0,Y 433.234,Z 377.081,A -85,B 0,C 180,E1 19771.613,E2 19771.613} C_VEL
LIN {X 0,Y 433.283,Z 377.552,A -85,B 0,C 180,E1 19770.503,E2 19770.503} C_VEL
LIN {X 0,Y 435.126,Z 381.361,A -85,B 0,C 180,E1 19769.328,E2 19769.328} C_VEL
LIN {X 0,Y 436.628,Z 383.246,A -85,B 0,C 180,E1 19768.757,E2 19768.757} C_VEL
LIN {X 0,Y 439.865,Z 387.507,A -85,B 0,C 180,E1 19767.789,E2 19767.789} C_VEL
LIN {X 0,Y 441.851,Z 390.07,A -85,B 0,C 180,E1 19767.222,E2 19767.222} C_VEL
LIN {X 0,Y 445.725,Z 395.25,A -85,B 0,C 180,E1 19766.16,E2 19766.16} C_VEL
LIN {X 0,Y 449.738,Z 400.575,A -85,B 0,C 180,E1 19765.155,E2 19765.155} C_VEL
LIN {X 0,Y 456.895,Z 410.607,A -85,B 0,C 180,E1 19763.471,E2 19763.471} C_VEL
LIN {X 0,Y 466.157,Z 424.544,A -85,B 0,C 180,E1 19761.498,E2 19761.498} C_VEL
LIN {X 0,Y 476.567,Z 441.492,A -85,B 0,C 180,E1 19759.489,E2 19759.489} C_VEL
LIN {X 0,Y 477.468,Z 443.422,A -85,B 0,C 180,E1 19759.314,E2 19759.314} C_VEL
LIN {X 0,Y 470.667,Z 640.445,A -85,B 0,C 180,E1 19755.736,E2 19755.736} C_VEL
LIN {X 0,Y 467.506,Z 738.805,A -85,B 0,C 180,E1 19753.969,E2 19753.969} C_VEL
LIN {X 0,Y 465.807,Z 762.117,A -85,B 0,C 180,E1 19753.363,E2 19753.363} C_VEL
LIN {X 0,Y 463.787,Z 784.656,A -85,B 0,C 180,E1 19752.565,E2 19752.565} C_VEL
LIN {X 0,Y 461.479,Z 805.133,A -85,B 0,C 180,E1 19751.627,E2 19751.627} C_VEL
LIN {X 0,Y 458.754,Z 826.784,A -85,B 0,C 180,E1 19750.424,E2 19750.424} C_VEL
LIN {X 0,Y 455.763,Z 847.396,A -85,B 0,C 180,E1 19749.025,E2 19749.025} C_VEL
LIN {X 0,Y 452.48,Z 868.811,A -85,B 0,C 180,E1 19747.298,E2 19747.298} C_VEL
LIN {X 0,Y 449.625,Z 886.345,A -85,B 0,C 180,E1 19745.638,E2 19745.638} C_VEL
LIN {X 0,Y 446.267,Z 906.224,A -85,B 0,C 180,E1 19743.449,E2 19743.449} C_VEL
LIN {X 0,Y 443.458,Z 923.101,A -85,B 0,C 180,E1 19741.293,E2 19741.293} C_VEL
LIN {X 0,Y 440.719,Z 939.385,A -85,B 0,C 180,E1 19738.871,E2 19738.871} C_VEL
LIN {X 0,Y 438.396,Z 954.309,A -85,B 0,C 180,E1 19736.322,E2 19736.322} C_VEL
LIN {X 0,Y 436.503,Z 967.051,A -85,B 0,C 180,E1 19733.778,E2 19733.778} C_VEL
LIN {X 0,Y 434.819,Z 979.276,A -85,B 0,C 180,E1 19730.883,E2 19730.883} C_VEL
LIN {X 0,Y 433.663,Z 989.048,A -85,B 0,C 180,E1 19728.138,E2 19728.138} C_VEL
LIN {X 0,Y 432.78,Z 998.337,A -85,B 0,C 180,E1 19724.999,E2 19724.999} C_VEL
LIN {X 0,Y 432.321,Z 1004.856,A -85,B 0,C 180,E1 19722.288,E2 19722.288} C_VEL
LIN {X 0,Y 432.047,Z 1010.631,A -85,B 0,C 180,E1 19719.192,E2 19719.192} C_VEL
LIN {X 0,Y 431.947,Z 1014.274,A -85,B 0,C 180,E1 19716.516,E2 19716.516} C_VEL
LIN {X 0,Y 431.89,Z 1016.914,A -85,B 0,C 180,E1 19713.454,E2 19713.454} C_VEL
LIN {X 0,Y 431.89,Z 1017.848,A -85,B 0,C 180,E1 19710.932,E2 19710.932} C_VEL
LIN {X 0,Y 431.907,Z 1017.69,A -85,B 0,C 180,E1 19708.146,E2 19708.146} C_VEL
LIN {X 0,Y 431.91,Z 1015.957,A -85,B 0,C 180,E1 19705.223,E2 19705.223} C_VEL
LIN {X 0,Y 431.946,Z 1013.164,A -85,B 0,C 180,E1 19702.556,E2 19702.556} C_VEL
LIN {X 0,Y 432.128,Z 1008.343,A -85,B 0,C 180,E1 19699.472,E2 19699.472} C_VEL
LIN {X 0,Y 432.462,Z 1002.683,A -85,B 0,C 180,E1 19696.743,E2 19696.743} C_VEL
LIN {X 0,Y 433.106,Z 994.562,A -85,B 0,C 180,E1 19693.646,E2 19693.646} C_VEL
LIN {X 0,Y 434.021,Z 985.864,A -85,B 0,C 180,E1 19690.91,E2 19690.91} C_VEL
LIN {X 0,Y 435.392,Z 974.879,A -85,B 0,C 180,E1 19688.022,E2 19688.022} C_VEL
LIN {X 0,Y 436.906,Z 964.22,A -85,B 0,C 180,E1 19685.618,E2 19685.618} C_VEL
LIN {X 0,Y 439.055,Z 950.074,A -85,B 0,C 180,E1 19682.91,E2 19682.91} C_VEL
LIN {X 0,Y 441.533,Z 935.013,A -85,B 0,C 180,E1 19680.408,E2 19680.408} C_VEL
LIN {X 0,Y 444.321,Z 918.299,A -85,B 0,C 180,E1 19678.033,E2 19678.033} C_VEL
LIN {X 0,Y 447.455,Z 900.204,A -85,B 0,C 180,E1 19675.804,E2 19675.804} C_VEL
LIN {X 0,Y 450.366,Z 882.871,A -85,B 0,C 180,E1 19673.967,E2 19673.967} C_VEL
LIN {X 0,Y 453.77,Z 862.029,A -85,B 0,C 180,E1 19672.071,E2 19672.071} C_VEL
LIN {X 0,Y 456.726,Z 842.915,A -85,B 0,C 180,E1 19670.596,E2 19670.596} C_VEL
LIN {X 0,Y 459.787,Z 820.959,A -85,B 0,C 180,E1 19669.179,E2 19669.179} C_VEL
LIN {X 0,Y 462.419,Z 799.937,A -85,B 0,C 180,E1 19668.056,E2 19668.056} C_VEL
LIN {X 0,Y 464.775,Z 777.412,A -85,B 0,C 180,E1 19667.11,E2 19667.11} C_VEL
LIN {X 0,Y 466.776,Z 754.471,A -85,B 0,C 180,E1 19666.37,E2 19666.37} C_VEL
LIN {X 0,Y 468.078,Z 731.92,A -85,B 0,C 180,E1 19665.86,E2 19665.86} C_VEL
LIN {X 0,Y 474.721,Z 520.938,A -85,B 0,C 180,E1 19662.101,E2 19662.101} C_VEL
LIN {X 0,Y 477.275,Z 443.062,A -85,B 0,C 180,E1 19660.681,E2 19660.681} C_VEL
LIN {X 0,Y 466.077,Z 425.492,A -85,B 0,C 180,E1 19658.664,E2 19658.664} C_VEL
LIN {X 0,Y 455.692,Z 410.555,A -85,B 0,C 180,E1 19656.68,E2 19656.68} C_VEL
LIN {X 0,Y 445.6,Z 396.628,A -85,B 0,C 180,E1 19654.589,E2 19654.589} C_VEL
LIN {X 0,Y 441.419,Z 391.061,A -85,B 0,C 180,E1 19653.668,E2 19653.668} C_VEL
LIN {X 0,Y 437.701,Z 386.086,A -85,B 0,C 180,E1 19652.802,E2 19652.802} C_VEL
LIN {X 0,Y 435.571,Z 381.852,A -85,B 0,C 180,E1 19651.868,E2 19651.868} C_VEL
LIN {X 0,Y 433.616,Z 378.845,A -85,B 0,C 180,E1 19651.098,E2 19651.098} C_VEL
LIN {X 0,Y 433.213,Z 377.266,A -85,B 0,C 180,E1 19650.668,E2 19650.668} C_VEL
LIN {X 0,Y 433.187,Z 377.09,A -85,B 0,C 180,E1 19647.309,E2 19647.309} C_VEL
LIN {X 0,Y 433.223,Z 377.074,A -85,B 0,C 180,E1 19643.629,E2 19643.629} C_VEL
LIN {X 0,Y 433.217,Z 377.076,A -85,B 0,C 180,E1 19639.973,E2 19639.973} C_VEL
LIN {X 0,Y 433.188,Z 377.084,A -85,B 0,C 180,E1 19636.355,E2 19636.355} C_VEL
LIN {X 0,Y 433.189,Z 377.088,A -85,B 0,C 180,E1 19632.53,E2 19632.53} C_VEL
LIN {X 0,Y 433.202,Z 377.081,A -85,B 0,C 180,E1 19628.762,E2 19628.762} C_VEL
LIN {X 0,Y 433.241,Z 377.072,A -85,B 0,C 180,E1 19625.164,E2 19625.164} C_VEL
LIN {X 0,Y 433.243,Z 377.071,A -85,B 0,C 180,E1 19621.322,E2 19621.322} C_VEL
LIN {X 0,Y 433.205,Z 377.075,A -85,B 0,C 180,E1 19617.751,E2 19617.751} C_VEL
LIN {X 0,Y 433.201,Z 377.073,A -85,B 0,C 180,E1 19614.038,E2 19614.038} C_VEL
LIN {X 0,Y 433.228,Z 377.073,A -85,B 0,C 180,E1 19610.434,E2 19610.434} C_VEL
LIN {X 0,Y 433.257,Z 377.071,A -85,B 0,C 180,E1 19606.657,E2 19606.657} C_VEL
LIN {X 0,Y 433.24,Z 377.072,A -85,B 0,C 180,E1 19602.956,E2 19602.956} C_VEL
LIN {X 0,Y 433.217,Z 377.074,A -85,B 0,C 180,E1 19599.321,E2 19599.321} C_VEL
LIN {X 0,Y 433.218,Z 377.078,A -85,B 0,C 180,E1 19595.598,E2 19595.598} C_VEL
LIN {X 0,Y 433.244,Z 377.078,A -85,B 0,C 180,E1 19591.913,E2 19591.913} C_VEL
LIN {X 0,Y 433.263,Z 377.076,A -85,B 0,C 180,E1 19588.253,E2 19588.253} C_VEL
LIN {X 0,Y 433.249,Z 377.081,A -85,B 0,C 180,E1 19584.439,E2 19584.439} C_VEL
LIN {X 0,Y 433.234,Z 377.084,A -85,B 0,C 180,E1 19580.629,E2 19580.629} C_VEL
LIN {X 0,Y 433.229,Z 377.078,A -85,B 0,C 180,E1 19576.821,E2 19576.821} C_VEL
LIN {X 0,Y 433.232,Z 377.071,A -85,B 0,C 180,E1 19572.978,E2 19572.978} C_VEL
LIN {X 0,Y 433.254,Z 377.077,A -85,B 0,C 180,E1 19569.216,E2 19569.216} C_VEL
LIN {X 0,Y 433.258,Z 377.078,A -85,B 0,C 180,E1 19565.392,E2 19565.392} C_VEL
LIN {X 0,Y 433.255,Z 377.048,A -85,B 0,C 180,E1 19561.587,E2 19561.587} C_VEL
LIN {X 0,Y 433.256,Z 377.078,A -85,B 0,C 180,E1 19557.781,E2 19557.781} C_VEL
LIN {X 0,Y 433.277,Z 377.269,A -85,B 0,C 180,E1 19555.843,E2 19555.843} C_VEL
LIN {X 0,Y 433.626,Z 378.653,A -85,B 0,C 180,E1 19555.538,E2 19555.538} C_VEL
LIN {X 0,Y 435.48,Z 381.657,A -85,B 0,C 180,E1 19555.072,E2 19555.072} C_VEL
LIN {X 0,Y 437.878,Z 383.745,A -85,B 0,C 180,E1 19554.551,E2 19554.551} C_VEL
LIN {X 0,Y 440.369,Z 387.558,A -85,B 0,C 180,E1 19553.975,E2 19553.975} C_VEL
LIN {X 0,Y 442.549,Z 389.707,A -85,B 0,C 180,E1 19553.517,E2 19553.517} C_VEL
LIN {X 0,Y 445.732,Z 393.951,A -85,B 0,C 180,E1 19552.83,E2 19552.83} C_VEL
LIN {X 0,Y 447.404,Z 395.994,A -85,B 0,C 180,E1 19552.479,E2 19552.479} C_VEL
LIN {X 0,Y 452.487,Z 402.704,A -85,B 0,C 180,E1 19551.425,E2 19551.425} C_VEL
LIN {X 0,Y 459.961,Z 412.46,A -85,B 0,C 180,E1 19549.964,E2 19549.964} C_VEL
LIN {X 0,Y 472.427,Z 429.593,A -85,B 0,C 180,E1 19547.695,E2 19547.695} C_VEL
LIN {X 0,Y 477.052,Z 436.789,A -85,B 0,C 180,E1 19546.884,E2 19546.884} C_VEL
LIN {X 0,Y 476.02,Z 466.557,A -85,B 0,C 180,E1 19546.345,E2 19546.345} C_VEL
LIN {X 0,Y 475.091,Z 474.256,A -85,B 0,C 180,E1 19546.295,E2 19546.295} C_VEL
LIN {X 0,Y 470.167,Z 494.869,A -85,B 0,C 180,E1 19546.49,E2 19546.49} C_VEL
LIN {X 0,Y 469.426,Z 501.475,A -85,B 0,C 180,E1 19546.439,E2 19546.439} C_VEL
LIN {X 0,Y 462.422,Z 708.058,A -85,B 0,C 180,E1 19542.714,E2 19542.714} C_VEL
LIN {X 0,Y 460.971,Z 731.281,A -85,B 0,C 180,E1 19542.158,E2 19542.158} C_VEL
LIN {X 0,Y 458.978,Z 753.455,A -85,B 0,C 180,E1 19541.402,E2 19541.402} C_VEL
LIN {X 0,Y 456.492,Z 776.058,A -85,B 0,C 180,E1 19540.4,E2 19540.4} C_VEL
LIN {X 0,Y 453.908,Z 795.67,A -85,B 0,C 180,E1 19539.32,E2 19539.32} C_VEL
LIN {X 0,Y 450.713,Z 816.991,A -85,B 0,C 180,E1 19537.902,E2 19537.902} C_VEL
LIN {X 0,Y 447.593,Z 835.791,A -85,B 0,C 180,E1 19536.409,E2 19536.409} C_VEL
LIN {X 0,Y 444.011,Z 855.926,A -85,B 0,C 180,E1 19534.517,E2 19534.517} C_VEL
LIN {X 0,Y 440.677,Z 874.007,A -85,B 0,C 180,E1 19532.532,E2 19532.532} C_VEL
LIN {X 0,Y 437.28,Z 891.576,A -85,B 0,C 180,E1 19530.259,E2 19530.259} C_VEL
LIN {X 0,Y 434.122,Z 908.23,A -85,B 0,C 180,E1 19527.753,E2 19527.753} C_VEL
LIN {X 0,Y 431.338,Z 923.411,A -85,B 0,C 180,E1 19525.077,E2 19525.077} C_VEL
LIN {X 0,Y 428.93,Z 937.354,A -85,B 0,C 180,E1 19522.181,E2 19522.181} C_VEL
LIN {X 0,Y 427.058,Z 949.478,A -85,B 0,C 180,E1 19519.201,E2 19519.201} C_VEL
LIN {X 0,Y 425.649,Z 960.569,A -85,B 0,C 180,E1 19515.966,E2 19515.966} C_VEL
LIN {X 0,Y 424.821,Z 968.938,A -85,B 0,C 180,E1 19513.028,E2 19513.028} C_VEL
LIN {X 0,Y 424.293,Z 976.152,A -85,B 0,C 180,E1 19509.873,E2 19509.873} C_VEL
LIN {X 0,Y 424.011,Z 981.456,A -85,B 0,C 180,E1 19506.806,E2 19506.806} C_VEL
LIN {X 0,Y 423.911,Z 985.087,A -85,B 0,C 180,E1 19503.825,E2 19503.825} C_VEL
LIN {X 0,Y 423.92,Z 987.292,A -85,B 0,C 180,E1 19500.773,E2 19500.773} C_VEL
LIN {X 0,Y 423.904,Z 987.98,A -85,B 0,C 180,E1 19497.784,E2 19497.784} C_VEL
LIN {X 0,Y 423.914,Z 987.103,A -85,B 0,C 180,E1 19494.696,E2 19494.696} C_VEL
LIN {X 0,Y 423.929,Z 984.667,A -85,B 0,C 180,E1 19491.659,E2 19491.659} C_VEL
LIN {X 0,Y 424.066,Z 980.619,A -85,B 0,C 180,E1 19488.572,E2 19488.572} C_VEL
LIN {X 0,Y 424.357,Z 974.787,A -85,B 0,C 180,E1 19485.398,E2 19485.398} C_VEL
LIN {X 0,Y 424.93,Z 967.571,A -85,B 0,C 180,E1 19482.364,E2 19482.364} C_VEL
LIN {X 0,Y 425.868,Z 958.682,A -85,B 0,C 180,E1 19479.34,E2 19479.34} C_VEL
LIN {X 0,Y 427.392,Z 947.31,A -85,B 0,C 180,E1 19476.125,E2 19476.125} C_VEL
LIN {X 0,Y 429.358,Z 934.964,A -85,B 0,C 180,E1 19473.179,E2 19473.179} C_VEL
LIN {X 0,Y 431.847,Z 920.728,A -85,B 0,C 180,E1 19470.314,E2 19470.314} C_VEL
LIN {X 0,Y 434.726,Z 905.452,A -85,B 0,C 180,E1 19467.684,E2 19467.684} C_VEL
LIN {X 0,Y 437.759,Z 889.419,A -85,B 0,C 180,E1 19465.332,E2 19465.332} C_VEL
LIN {X 0,Y 441.304,Z 870.942,A -85,B 0,C 180,E1 19463.007,E2 19463.007} C_VEL
LIN {X 0,Y 444.463,Z 853.919,A -85,B 0,C 180,E1 19461.166,E2 19461.166} C_VEL
LIN {X 0,Y 447.921,Z 834.282,A -85,B 0,C 180,E1 19459.359,E2 19459.359} C_VEL
LIN {X 0,Y 451.218,Z 814.43,A -85,B 0,C 180,E1 19457.806,E2 19457.806} C_VEL
LIN {X 0,Y 454.132,Z 794.285,A -85,B 0,C 180,E1 19456.501,E2 19456.501} C_VEL
LIN {X 0,Y 456.89,Z 773.135,A -85,B 0,C 180,E1 19455.355,E2 19455.355} C_VEL
LIN {X 0,Y 459.214,Z 751.001,A -85,B 0,C 180,E1 19454.415,E2 19454.415} C_VEL
LIN {X 0,Y 461.245,Z 727.048,A -85,B 0,C 180,E1 19453.644,E2 19453.644} C_VEL
LIN {X 0,Y 462.497,Z 705.243,A -85,B 0,C 180,E1 19453.149,E2 19453.149} C_VEL
LIN {X 0,Y 469.817,Z 499.484,A -85,B 0,C 180,E1 19449.403,E2 19449.403} C_VEL
LIN {X 0,Y 472.051,Z 440.282,A -85,B 0,C 180,E1 19448.282,E2 19448.282} C_VEL
LIN {X 0,Y 461.389,Z 424.677,A -85,B 0,C 180,E1 19446.174,E2 19446.174} C_VEL
LIN {X 0,Y 452.764,Z 412.723,A -85,B 0,C 180,E1 19444.275,E2 19444.275} C_VEL
LIN {X 0,Y 447.94,Z 406.647,A -85,B 0,C 180,E1 19443.135,E2 19443.135} C_VEL
LIN {X 0,Y 444.404,Z 401.973,A -85,B 0,C 180,E1 19442.225,E2 19442.225} C_VEL
LIN {X 0,Y 440.942,Z 397.593,A -85,B 0,C 180,E1 19441.3,E2 19441.3} C_VEL
LIN {X 0,Y 439.195,Z 395.78,A -85,B 0,C 180,E1 19440.816,E2 19440.816} C_VEL
LIN {X 0,Y 436.275,Z 391.872,A -85,B 0,C 180,E1 19439.935,E2 19439.935} C_VEL
LIN {X 0,Y 435.428,Z 390.73,A -85,B 0,C 180,E1 19439.672,E2 19439.672} C_VEL
LIN {X 0,Y 432.378,Z 387.98,A -85,B 0,C 180,E1 19438.742,E2 19438.742} C_VEL
LIN {X 0,Y 430.591,Z 384.716,A -85,B 0,C 180,E1 19438.071,E2 19438.071} C_VEL
LIN {X 0,Y 427.212,Z 382.322,A -85,B 0,C 180,E1 19436.915,E2 19436.915} C_VEL
LIN {X 0,Y 425.472,Z 378.939,A -85,B 0,C 180,E1 19436.093,E2 19436.093} C_VEL
LIN {X 0,Y 425.302,Z 378.096,A -85,B 0,C 180,E1 19435.416,E2 19435.416} C_VEL
LIN {X 0,Y 425.297,Z 378.067,A -85,B 0,C 180,E1 19431.619,E2 19431.619} C_VEL
LIN {X 0,Y 425.302,Z 378.07,A -85,B 0,C 180,E1 19427.785,E2 19427.785} C_VEL
LIN {X 0,Y 425.318,Z 378.07,A -85,B 0,C 180,E1 19424.036,E2 19424.036} C_VEL
LIN {X 0,Y 425.318,Z 378.07,A -85,B 0,C 180,E1 19420.214,E2 19420.214} C_VEL
LIN {X 0,Y 425.293,Z 378.063,A -85,B 0,C 180,E1 19416.443,E2 19416.443} C_VEL
LIN {X 0,Y 425.297,Z 378.29,A -85,B 0,C 180,E1 19412.903,E2 19412.903} C_VEL
LIN {X 0,Y 426.49,Z 381.351,A -85,B 0,C 180,E1 19411.826,E2 19411.826} C_VEL
LIN {X 0,Y 429.804,Z 385.009,A -85,B 0,C 180,E1 19410.604,E2 19410.604} C_VEL
LIN {X 0,Y 433.273,Z 389.241,A -85,B 0,C 180,E1 19409.414,E2 19409.414} C_VEL
LIN {X 0,Y 437.813,Z 395.089,A -85,B 0,C 180,E1 19408.006,E2 19408.006} C_VEL
LIN {X 0,Y 443.254,Z 402.634,A -85,B 0,C 180,E1 19406.451,E2 19406.451} C_VEL
LIN {X 0,Y 446.973,Z 407.665,A -85,B 0,C 180,E1 19405.493,E2 19405.493} C_VEL
LIN {X 0,Y 455.123,Z 419.308,A -85,B 0,C 180,E1 19403.541,E2 19403.541} C_VEL
LIN {X 0,Y 465.637,Z 435.715,A -85,B 0,C 180,E1 19401.289,E2 19401.289} C_VEL
LIN {X 0,Y 472.193,Z 446.973,A -85,B 0,C 180,E1 19399.994,E2 19399.994} C_VEL
LIN {X 0,Y 464.968,Z 642.849,A -85,B 0,C 180,E1 19396.394,E2 19396.394} C_VEL
LIN {X 0,Y 461.676,Z 738.544,A -85,B 0,C 180,E1 19394.653,E2 19394.653} C_VEL
LIN {X 0,Y 459.866,Z 762.057,A -85,B 0,C 180,E1 19394.036,E2 19394.036} C_VEL
LIN {X 0,Y 457.711,Z 784.717,A -85,B 0,C 180,E1 19393.225,E2 19393.225} C_VEL
LIN {X 0,Y 455.217,Z 805.676,A -85,B 0,C 180,E1 19392.252,E2 19392.252} C_VEL
LIN {X 0,Y 452.339,Z 827.164,A -85,B 0,C 180,E1 19391.036,E2 19391.036} C_VEL
LIN {X 0,Y 449.235,Z 847.493,A -85,B 0,C 180,E1 19389.639,E2 19389.639} C_VEL
LIN {X 0,Y 445.805,Z 868.555,A -85,B 0,C 180,E1 19387.921,E2 19387.921} C_VEL
LIN {X 0,Y 442.723,Z 886.484,A -85,B 0,C 180,E1 19386.201,E2 19386.201} C_VEL
LIN {X 0,Y 439.278,Z 905.72,A -85,B 0,C 180,E1 19384.054,E2 19384.054} C_VEL
LIN {X 0,Y 436.299,Z 922.49,A -85,B 0,C 180,E1 19381.885,E2 19381.885} C_VEL
LIN {X 0,Y 433.391,Z 938.76,A -85,B 0,C 180,E1 19379.436,E2 19379.436} C_VEL
LIN {X 0,Y 430.959,Z 953.448,A -85,B 0,C 180,E1 19376.902,E2 19376.902} C_VEL
LIN {X 0,Y 428.84,Z 966.642,A -85,B 0,C 180,E1 19374.23,E2 19374.23} C_VEL
LIN {X 0,Y 427.139,Z 978.674,A -85,B 0,C 180,E1 19371.421,E2 19371.421} C_VEL
LIN {X 0,Y 425.932,Z 988.129,A -85,B 0,C 180,E1 19368.763,E2 19368.763} C_VEL
LIN {X 0,Y 424.976,Z 997.277,A -85,B 0,C 180,E1 19365.701,E2 19365.701} C_VEL
LIN {X 0,Y 424.401,Z 1004.25,A -85,B 0,C 180,E1 19362.798,E2 19362.798} C_VEL
LIN {X 0,Y 424.063,Z 1010.218,A -85,B 0,C 180,E1 19359.64,E2 19359.64} C_VEL
LIN {X 0,Y 423.936,Z 1013.955,A -85,B 0,C 180,E1 19356.912,E2 19356.912} C_VEL
LIN {X 0,Y 423.908,Z 1016.733,A -85,B 0,C 180,E1 19353.881,E2 19353.881} C_VEL
LIN {X 0,Y 423.897,Z 1017.825,A -85,B 0,C 180,E1 19351.085,E2 19351.085} C_VEL
LIN {X 0,Y 423.906,Z 1017.735,A -85,B 0,C 180,E1 19348.382,E2 19348.382} C_VEL
LIN {X 0,Y 423.909,Z 1016.071,A -85,B 0,C 180,E1 19345.268,E2 19345.268} C_VEL
LIN {X 0,Y 423.942,Z 1013.483,A -85,B 0,C 180,E1 19342.687,E2 19342.687} C_VEL
LIN {X 0,Y 424.11,Z 1009.106,A -85,B 0,C 180,E1 19339.682,E2 19339.682} C_VEL
LIN {X 0,Y 424.467,Z 1003.355,A -85,B 0,C 180,E1 19336.796,E2 19336.796} C_VEL
LIN {X 0,Y 425.145,Z 995.371,A -85,B 0,C 180,E1 19333.612,E2 19333.612} C_VEL
LIN {X 0,Y 426.096,Z 986.78,A -85,B 0,C 180,E1 19330.826,E2 19330.826} C_VEL
LIN {X 0,Y 427.446,Z 976.471,A -85,B 0,C 180,E1 19328.026,E2 19328.026} C_VEL
LIN {X 0,Y 429.141,Z 964.802,A -85,B 0,C 180,E1 19325.356,E2 19325.356} C_VEL
LIN {X 0,Y 431.46,Z 950.504,A -85,B 0,C 180,E1 19322.543,E2 19322.543} C_VEL
LIN {X 0,Y 433.9,Z 936.461,A -85,B 0,C 180,E1 19320.155,E2 19320.155} C_VEL
LIN {X 0,Y 436.882,Z 919.778,A -85,B 0,C 180,E1 19317.703,E2 19317.703} C_VEL
LIN {X 0,Y 440.141,Z 902.182,A -85,B 0,C 180,E1 19315.462,E2 19315.462} C_VEL
LIN {X 0,Y 443.394,Z 883.815,A -85,B 0,C 180,E1 19313.47,E2 19313.47} C_VEL
LIN {X 0,Y 446.848,Z 864.058,A -85,B 0,C 180,E1 19311.622,E2 19311.622} C_VEL
LIN {X 0,Y 449.92,Z 845.195,A -85,B 0,C 180,E1 19310.13,E2 19310.13} C_VEL
LIN {X 0,Y 453.099,Z 824.209,A -85,B 0,C 180,E1 19308.721,E2 19308.721} C_VEL
LIN {X 0,Y 455.806,Z 803.691,A -85,B 0,C 180,E1 19307.588,E2 19307.588} C_VEL
LIN {X 0,Y 458.519,Z 779.898,A -85,B 0,C 180,E1 19306.536,E2 19306.536} C_VEL
LIN {X 0,Y 460.542,Z 758.236,A -85,B 0,C 180,E1 19305.803,E2 19305.803} C_VEL
LIN {X 0,Y 462.126,Z 734.569,A -85,B 0,C 180,E1 19305.233,E2 19305.233} C_VEL
LIN {X 0,Y 469.122,Z 525.645,A -85,B 0,C 180,E1 19301.469,E2 19301.469} C_VEL
LIN {X 0,Y 471.829,Z 446.658,A -85,B 0,C 180,E1 19300.007,E2 19300.007} C_VEL
LIN {X 0,Y 461.046,Z 429.949,A -85,B 0,C 180,E1 19298.017,E2 19298.017} C_VEL
LIN {X 0,Y 452.008,Z 416.745,A -85,B 0,C 180,E1 19296.239,E2 19296.239} C_VEL
LIN {X 0,Y 442.041,Z 402.872,A -85,B 0,C 180,E1 19294.121,E2 19294.121} C_VEL
LIN {X 0,Y 438.015,Z 397.469,A -85,B 0,C 180,E1 19293.219,E2 19293.219} C_VEL
LIN {X 0,Y 434.289,Z 392.584,A -85,B 0,C 180,E1 19292.362,E2 19292.362} C_VEL
LIN {X 0,Y 430.285,Z 387.384,A -85,B 0,C 180,E1 19291.405,E2 19291.405} C_VEL
LIN {X 0,Y 428.457,Z 384.623,A -85,B 0,C 180,E1 19290.831,E2 19290.831} C_VEL
LIN {X 0,Y 427.305,Z 382.456,A -85,B 0,C 180,E1 19290.307,E2 19290.307} C_VEL
LIN {X 0,Y 425.441,Z 379.04,A -85,B 0,C 180,E1 19289.418,E2 19289.418} C_VEL
LIN {X 0,Y 425.257,Z 378.197,A -85,B 0,C 180,E1 19289.123,E2 19289.123} C_VEL
LIN {X 0,Y 425.265,Z 378.066,A -85,B 0,C 180,E1 19285.479,E2 19285.479} C_VEL
LIN {X 0,Y 425.3,Z 378.072,A -85,B 0,C 180,E1 19281.66,E2 19281.66} C_VEL
LIN {X 0,Y 425.289,Z 378.065,A -85,B 0,C 180,E1 19277.796,E2 19277.796} C_VEL
LIN {X 0,Y 425.255,Z 378.065,A -85,B 0,C 180,E1 19274.153,E2 19274.153} C_VEL
LIN {X 0,Y 425.252,Z 378.07,A -85,B 0,C 180,E1 19270.43,E2 19270.43} C_VEL
LIN {X 0,Y 425.26,Z 378.075,A -85,B 0,C 180,E1 19266.615,E2 19266.615} C_VEL
LIN {X 0,Y 425.293,Z 378.073,A -85,B 0,C 180,E1 19262.964,E2 19262.964} C_VEL
LIN {X 0,Y 425.315,Z 378.069,A -85,B 0,C 180,E1 19259.191,E2 19259.191} C_VEL
LIN {X 0,Y 425.294,Z 378.067,A -85,B 0,C 180,E1 19255.28,E2 19255.28} C_VEL
LIN {X 0,Y 425.272,Z 378.07,A -85,B 0,C 180,E1 19251.618,E2 19251.618} C_VEL
LIN {X 0,Y 425.269,Z 378.068,A -85,B 0,C 180,E1 19247.783,E2 19247.783} C_VEL
LIN {X 0,Y 425.281,Z 378.063,A -85,B 0,C 180,E1 19244.033,E2 19244.033} C_VEL
LIN {X 0,Y 425.311,Z 378.057,A -85,B 0,C 180,E1 19240.355,E2 19240.355} C_VEL
LIN {X 0,Y 425.319,Z 378.058,A -85,B 0,C 180,E1 19236.591,E2 19236.591} C_VEL
LIN {X 0,Y 425.292,Z 378.061,A -85,B 0,C 180,E1 19232.864,E2 19232.864} C_VEL
LIN {X 0,Y 425.281,Z 378.06,A -85,B 0,C 180,E1 19229.097,E2 19229.097} C_VEL
LIN {X 0,Y 425.286,Z 378.064,A -85,B 0,C 180,E1 19225.323,E2 19225.323} C_VEL
LIN {X 0,Y 425.303,Z 378.069,A -85,B 0,C 180,E1 19221.515,E2 19221.515} C_VEL
LIN {X 0,Y 425.321,Z 378.069,A -85,B 0,C 180,E1 19217.752,E2 19217.752} C_VEL
LIN {X 0,Y 425.319,Z 378.063,A -85,B 0,C 180,E1 19213.901,E2 19213.901} C_VEL
LIN {X 0,Y 425.315,Z 378.06,A -85,B 0,C 180,E1 19210.095,E2 19210.095} C_VEL
LIN {X 0,Y 425.302,Z 378.067,A -85,B 0,C 180,E1 19206.256,E2 19206.256} C_VEL
LIN {X 0,Y 425.298,Z 378.058,A -85,B 0,C 180,E1 19202.407,E2 19202.407} C_VEL
LIN {X 0,Y 425.305,Z 378.057,A -85,B 0,C 180,E1 19198.5,E2 19198.5} C_VEL
LIN {X 0,Y 425.356,Z 378.331,A -85,B 0,C 180,E1 19197.429,E2 19197.429} C_VEL
LIN {X 0,Y 425.749,Z 379.826,A -85,B 0,C 180,E1 19197.117,E2 19197.117} C_VEL
LIN {X 0,Y 427.715,Z 382.832,A -85,B 0,C 180,E1 19196.599,E2 19196.599} C_VEL
LIN {X 0,Y 430.032,Z 384.646,A -85,B 0,C 180,E1 19196.063,E2 19196.063} C_VEL
LIN {X 0,Y 432.413,Z 388.427,A -85,B 0,C 180,E1 19195.468,E2 19195.468} C_VEL
LIN {X 0,Y 434.818,Z 390.855,A -85,B 0,C 180,E1 19194.924,E2 19194.924} C_VEL
LIN {X 0,Y 437.951,Z 395.049,A -85,B 0,C 180,E1 19194.206,E2 19194.206} C_VEL
LIN {X 0,Y 439.751,Z 397.188,A -85,B 0,C 180,E1 19193.811,E2 19193.811} C_VEL
LIN {X 0,Y 444.587,Z 403.353,A -85,B 0,C 180,E1 19192.768,E2 19192.768} C_VEL
LIN {X 0,Y 452.324,Z 413.426,A -85,B 0,C 180,E1 19191.168,E2 19191.168} C_VEL
LIN {X 0,Y 462.938,Z 427.858,A -85,B 0,C 180,E1 19189.124,E2 19189.124} C_VEL
LIN {X 0,Y 471.642,Z 440.521,A -85,B 0,C 180,E1 19187.548,E2 19187.548} C_VEL
LIN {X 0,Y 469.426,Z 501.475,A -85,B 0,C 180,E1 19186.439,E2 19186.439} C_VEL
LIN {X 0,Y 468.472,Z 509.176,A -85,B 0,C 180,E1 19186.392,E2 19186.392} C_VEL
LIN {X 0,Y 463.503,Z 529.777,A -85,B 0,C 180,E1 19186.592,E2 19186.592} C_VEL
LIN {X 0,Y 462.784,Z 536.379,A -85,B 0,C 180,E1 19186.537,E2 19186.537} C_VEL
LIN {X 0,Y 456.466,Z 712.965,A -85,B 0,C 180,E1 19183.317,E2 19183.317} C_VEL
LIN {X 0,Y 454.756,Z 736.27,A -85,B 0,C 180,E1 19182.701,E2 19182.701} C_VEL
LIN {X 0,Y 452.633,Z 758.656,A -85,B 0,C 180,E1 19181.894,E2 19181.894} C_VEL
LIN {X 0,Y 449.985,Z 780.127,A -85,B 0,C 180,E1 19180.883,E2 19180.883} C_VEL
LIN {X 0,Y 447.142,Z 800.513,A -85,B 0,C 180,E1 19179.716,E2 19179.716} C_VEL
LIN {X 0,Y 443.797,Z 820.93,A -85,B 0,C 180,E1 19178.287,E2 19178.287} C_VEL
LIN {X 0,Y 440.202,Z 841.415,A -85,B 0,C 180,E1 19176.583,E2 19176.583} C_VEL
LIN {X 0,Y 436.862,Z 858.98,A -85,B 0,C 180,E1 19174.854,E2 19174.854} C_VEL
LIN {X 0,Y 433.03,Z 878.237,A -85,B 0,C 180,E1 19172.643,E2 19172.643} C_VEL
LIN {X 0,Y 429.855,Z 894.008,A -85,B 0,C 180,E1 19170.53,E2 19170.53} C_VEL
LIN {X 0,Y 426.543,Z 910.341,A -85,B 0,C 180,E1 19167.982,E2 19167.982} C_VEL
LIN {X 0,Y 423.649,Z 925.318,A -85,B 0,C 180,E1 19165.258,E2 19165.258} C_VEL
LIN {X 0,Y 421.171,Z 938.824,A -85,B 0,C 180,E1 19162.357,E2 19162.357} C_VEL
LIN {X 0,Y 419.182,Z 950.93,A -85,B 0,C 180,E1 19159.274,E2 19159.274} C_VEL
LIN {X 0,Y 417.758,Z 961.183,A -85,B 0,C 180,E1 19156.149,E2 19156.149} C_VEL
LIN {X 0,Y 416.829,Z 969.753,A -85,B 0,C 180,E1 19152.981,E2 19152.981} C_VEL
LIN {X 0,Y 416.304,Z 976.528,A -85,B 0,C 180,E1 19149.899,E2 19149.899} C_VEL
LIN {X 0,Y 416.013,Z 981.753,A -85,B 0,C 180,E1 19146.783,E2 19146.783} C_VEL
LIN {X 0,Y 415.913,Z 985.125,A -85,B 0,C 180,E1 19143.897,E2 19143.897} C_VEL
LIN {X 0,Y 415.919,Z 987.315,A -85,B 0,C 180,E1 19140.768,E2 19140.768} C_VEL
LIN {X 0,Y 415.902,Z 987.975,A -85,B 0,C 180,E1 19137.741,E2 19137.741} C_VEL
LIN {X 0,Y 415.913,Z 987.158,A -85,B 0,C 180,E1 19134.76,E2 19134.76} C_VEL
LIN {X 0,Y 415.921,Z 984.942,A -85,B 0,C 180,E1 19131.823,E2 19131.823} C_VEL
LIN {X 0,Y 416.046,Z 981.222,A -85,B 0,C 180,E1 19128.783,E2 19128.783} C_VEL
LIN {X 0,Y 416.344,Z 975.857,A -85,B 0,C 180,E1 19125.663,E2 19125.663} C_VEL
LIN {X 0,Y 416.91,Z 968.864,A -85,B 0,C 180,E1 19122.556,E2 19122.556} C_VEL
LIN {X 0,Y 417.918,Z 959.993,A -85,B 0,C 180,E1 19119.347,E2 19119.347} C_VEL
LIN {X 0,Y 419.371,Z 949.801,A -85,B 0,C 180,E1 19116.304,E2 19116.304} C_VEL
LIN {X 0,Y 421.338,Z 938.026,A -85,B 0,C 180,E1 19113.348,E2 19113.348} C_VEL
LIN {X 0,Y 423.851,Z 924.575,A -85,B 0,C 180,E1 19110.477,E2 19110.477} C_VEL
LIN {X 0,Y 426.594,Z 910.418,A -85,B 0,C 180,E1 19107.914,E2 19107.914} C_VEL
LIN {X 0,Y 429.964,Z 893.869,A -85,B 0,C 180,E1 19105.334,E2 19105.334} C_VEL
LIN {X 0,Y 433.244,Z 877.708,A -85,B 0,C 180,E1 19103.172,E2 19103.172} C_VEL
LIN {X 0,Y 436.915,Z 859.219,A -85,B 0,C 180,E1 19101.057,E2 19101.057} C_VEL
LIN {X 0,Y 440.33,Z 841.287,A -85,B 0,C 180,E1 19099.293,E2 19099.293} C_VEL
LIN {X 0,Y 443.822,Z 821.379,A -85,B 0,C 180,E1 19097.641,E2 19097.641} C_VEL
LIN {X 0,Y 447.096,Z 801.361,A -85,B 0,C 180,E1 19096.233,E2 19096.233} C_VEL
LIN {X 0,Y 450.01,Z 780.479,A -85,B 0,C 180,E1 19095.035,E2 19095.035} C_VEL
LIN {X 0,Y 452.65,Z 758.856,A -85,B 0,C 180,E1 19094.018,E2 19094.018} C_VEL
LIN {X 0,Y 454.729,Z 736.971,A -85,B 0,C 180,E1 19093.228,E2 19093.228} C_VEL
LIN {X 0,Y 456.42,Z 713.598,A -85,B 0,C 180,E1 19092.608,E2 19092.608} C_VEL
LIN {X 0,Y 464.627,Z 500.114,A -85,B 0,C 180,E1 19088.66,E2 19088.66} C_VEL
LIN {X 0,Y 466.904,Z 444.424,A -85,B 0,C 180,E1 19087.599,E2 19087.599} C_VEL
LIN {X 0,Y 456.465,Z 428.883,A -85,B 0,C 180,E1 19085.437,E2 19085.437} C_VEL
LIN {X 0,Y 448.516,Z 418.08,A -85,B 0,C 180,E1 19083.614,E2 19083.614} C_VEL
LIN {X 0,Y 444.873,Z 413.276,A -85,B 0,C 180,E1 19082.706,E2 19082.706} C_VEL
LIN {X 0,Y 441.325,Z 408.632,A -85,B 0,C 180,E1 19081.771,E2 19081.771} C_VEL
LIN {X 0,Y 437.359,Z 403.536,A -85,B 0,C 180,E1 19080.655,E2 19080.655} C_VEL
LIN {X 0,Y 433.958,Z 399.346,A -85,B 0,C 180,E1 19079.629,E2 19079.629} C_VEL
LIN {X 0,Y 432.844,Z 397.93,A -85,B 0,C 180,E1 19079.279,E2 19079.279} C_VEL
LIN {X 0,Y 429.756,Z 394.679,A -85,B 0,C 180,E1 19078.267,E2 19078.267} C_VEL
LIN {X 0,Y 428.292,Z 392.121,A -85,B 0,C 180,E1 19077.709,E2 19077.709} C_VEL
LIN {X 0,Y 425.047,Z 389.568,A -85,B 0,C 180,E1 19076.561,E2 19076.561} C_VEL
LIN {X 0,Y 422.913,Z 385.84,A -85,B 0,C 180,E1 19075.594,E2 19075.594} C_VEL
LIN {X 0,Y 419.247,Z 383.282,A -85,B 0,C 180,E1 19074.003,E2 19074.003} C_VEL
LIN {X 0,Y 417.665,Z 380.441,A -85,B 0,C 180,E1 19073.057,E2 19073.057} C_VEL
LIN {X 0,Y 417.415,Z 379.274,A -85,B 0,C 180,E1 19072.43,E2 19072.43} C_VEL
LIN {X 0,Y 417.373,Z 379.059,A -85,B 0,C 180,E1 19068.672,E2 19068.672} C_VEL
LIN {X 0,Y 417.353,Z 379.06,A -85,B 0,C 180,E1 19064.863,E2 19064.863} C_VEL
LIN {X 0,Y 417.342,Z 379.062,A -85,B 0,C 180,E1 19061.13,E2 19061.13} C_VEL
LIN {X 0,Y 417.337,Z 379.065,A -85,B 0,C 180,E1 19057.282,E2 19057.282} C_VEL
LIN {X 0,Y 417.428,Z 379.447,A -85,B 0,C 180,E1 19055.821,E2 19055.821} C_VEL
LIN {X 0,Y 417.789,Z 380.893,A -85,B 0,C 180,E1 19055.279,E2 19055.279} C_VEL
LIN {X 0,Y 419.614,Z 383.697,A -85,B 0,C 180,E1 19054.254,E2 19054.254} C_VEL
LIN {X 0,Y 422.644,Z 386.144,A -85,B 0,C 180,E1 19052.91,E2 19052.91} C_VEL
LIN {X 0,Y 426.464,Z 391.031,A -85,B 0,C 180,E1 19051.351,E2 19051.351} C_VEL
LIN {X 0,Y 428.034,Z 392.99,A -85,B 0,C 180,E1 19050.778,E2 19050.778} C_VEL
LIN {X 0,Y 431.843,Z 397.721,A -85,B 0,C 180,E1 19049.456,E2 19049.456} C_VEL
LIN {X 0,Y 436.652,Z 404.189,A -85,B 0,C 180,E1 19047.95,E2 19047.95} C_VEL
LIN {X 0,Y 443.227,Z 413.218,A -85,B 0,C 180,E1 19046.099,E2 19046.099} C_VEL
LIN {X 0,Y 452.122,Z 426.344,A -85,B 0,C 180,E1 19043.889,E2 19043.889} C_VEL
LIN {X 0,Y 461.78,Z 441.607,A -85,B 0,C 180,E1 19041.759,E2 19041.759} C_VEL
LIN {X 0,Y 466.996,Z 450.781,A -85,B 0,C 180,E1 19040.686,E2 19040.686} C_VEL
LIN {X 0,Y 459.401,Z 643.688,A -85,B 0,C 180,E1 19037.1,E2 19037.1} C_VEL
LIN {X 0,Y 455.927,Z 738.378,A -85,B 0,C 180,E1 19035.354,E2 19035.354} C_VEL
LIN {X 0,Y 454.021,Z 761.892,A -85,B 0,C 180,E1 19034.731,E2 19034.731} C_VEL
LIN {X 0,Y 451.7,Z 784.81,A -85,B 0,C 180,E1 19033.902,E2 19033.902} C_VEL
LIN {X 0,Y 449.128,Z 805.32,A -85,B 0,C 180,E1 19032.942,E2 19032.942} C_VEL
LIN {X 0,Y 445.983,Z 827.596,A -85,B 0,C 180,E1 19031.664,E2 19031.664} C_VEL
LIN {X 0,Y 442.848,Z 847.106,A -85,B 0,C 180,E1 19030.308,E2 19030.308} C_VEL
LIN {X 0,Y 439.248,Z 867.988,A -85,B 0,C 180,E1 19028.59,E2 19028.59} C_VEL
LIN {X 0,Y 435.864,Z 886.624,A -85,B 0,C 180,E1 19026.781,E2 19026.781} C_VEL
LIN {X 0,Y 432.235,Z 905.786,A -85,B 0,C 180,E1 19024.606,E2 19024.606} C_VEL
LIN {X 0,Y 428.983,Z 923.06,A -85,B 0,C 180,E1 19022.334,E2 19022.334} C_VEL
LIN {X 0,Y 425.922,Z 939.175,A -85,B 0,C 180,E1 19019.849,E2 19019.849} C_VEL
LIN {X 0,Y 423.209,Z 954.46,A -85,B 0,C 180,E1 19017.131,E2 19017.131} C_VEL
LIN {X 0,Y 421.103,Z 966.88,A -85,B 0,C 180,E1 19014.555,E2 19014.555} C_VEL
LIN {X 0,Y 419.221,Z 979.384,A -85,B 0,C 180,E1 19011.541,E2 19011.541} C_VEL
LIN {X 0,Y 417.987,Z 988.87,A -85,B 0,C 180,E1 19008.843,E2 19008.843} C_VEL
LIN {X 0,Y 417.038,Z 997.629,A -85,B 0,C 180,E1 19005.865,E2 19005.865} C_VEL
LIN {X 0,Y 416.452,Z 1004.249,A -85,B 0,C 180,E1 19003.046,E2 19003.046} C_VEL
LIN {X 0,Y 416.074,Z 1010.218,A -85,B 0,C 180,E1 18999.827,E2 18999.827} C_VEL
LIN {X 0,Y 415.938,Z 1013.795,A -85,B 0,C 180,E1 18997.184,E2 18997.184} C_VEL
LIN {X 0,Y 415.91,Z 1016.519,A -85,B 0,C 180,E1 18994.277,E2 18994.277} C_VEL
LIN {X 0,Y 415.903,Z 1017.802,A -85,B 0,C 180,E1 18991.243,E2 18991.243} C_VEL
LIN {X 0,Y 415.907,Z 1017.758,A -85,B 0,C 180,E1 18988.488,E2 18988.488} C_VEL
LIN {X 0,Y 415.909,Z 1016.184,A -85,B 0,C 180,E1 18985.315,E2 18985.315} C_VEL
LIN {X 0,Y 415.943,Z 1013.643,A -85,B 0,C 180,E1 18982.684,E2 18982.684} C_VEL
LIN {X 0,Y 416.106,Z 1009.605,A -85,B 0,C 180,E1 18979.762,E2 18979.762} C_VEL
LIN {X 0,Y 416.498,Z 1003.658,A -85,B 0,C 180,E1 18976.68,E2 18976.68} C_VEL
LIN {X 0,Y 417.184,Z 996.18,A -85,B 0,C 180,E1 18973.576,E2 18973.576} C_VEL
LIN {X 0,Y 418.157,Z 987.51,A -85,B 0,C 180,E1 18970.737,E2 18970.737} C_VEL
LIN {X 0,Y 419.637,Z 976.722,A -85,B 0,C 180,E1 18967.743,E2 18967.743} C_VEL
LIN {X 0,Y 421.459,Z 964.956,A -85,B 0,C 180,E1 18964.991,E2 18964.991} C_VEL
LIN {X 0,Y 424.016,Z 950.147,A -85,B 0,C 180,E1 18962.019,E2 18962.019} C_VEL
LIN {X 0,Y 426.64,Z 936.075,A -85,B 0,C 180,E1 18959.59,E2 18959.59} C_VEL
LIN {X 0,Y 429.782,Z 919.527,A -85,B 0,C 180,E1 18957.122,E2 18957.122} C_VEL
LIN {X 0,Y 433.243,Z 901.918,A -85,B 0,C 180,E1 18954.85,E2 18954.85} C_VEL
LIN {X 0,Y 436.707,Z 883.401,A -85,B 0,C 180,E1 18952.817,E2 18952.817} C_VEL
LIN {X 0,Y 440.405,Z 863.429,A -85,B 0,C 180,E1 18950.936,E2 18950.936} C_VEL
LIN {X 0,Y 443.559,Z 844.982,A -85,B 0,C 180,E1 18949.465,E2 18949.465} C_VEL
LIN {X 0,Y 446.935,Z 823.654,A -85,B 0,C 180,E1 18948.024,E2 18948.024} C_VEL
LIN {X 0,Y 449.782,Z 803.107,A -85,B 0,C 180,E1 18946.883,E2 18946.883} C_VEL
LIN {X 0,Y 452.666,Z 778.995,A -85,B 0,C 180,E1 18945.818,E2 18945.818} C_VEL
LIN {X 0,Y 454.802,Z 757.187,A -85,B 0,C 180,E1 18945.083,E2 18945.083} C_VEL
LIN {X 0,Y 456.401,Z 733.723,A -85,B 0,C 180,E1 18944.52,E2 18944.52} C_VEL
LIN {X 0,Y 463.811,Z 523.807,A -85,B 0,C 180,E1 18940.703,E2 18940.703} C_VEL
LIN {X 0,Y 466.509,Z 450.468,A -85,B 0,C 180,E1 18939.336,E2 18939.336} C_VEL
LIN {X 0,Y 454.329,Z 431.543,A -85,B 0,C 180,E1 18937.006,E2 18937.006} C_VEL
LIN {X 0,Y 441.915,Z 413.712,A -85,B 0,C 180,E1 18934.407,E2 18934.407} C_VEL
LIN {X 0,Y 434.364,Z 403.542,A -85,B 0,C 180,E1 18932.708,E2 18932.708} C_VEL
LIN {X 0,Y 430.934,Z 399.019,A -85,B 0,C 180,E1 18931.899,E2 18931.899} C_VEL
LIN {X 0,Y 426.514,Z 393.24,A -85,B 0,C 180,E1 18930.811,E2 18930.811} C_VEL
LIN {X 0,Y 422.985,Z 388.687,A -85,B 0,C 180,E1 18929.918,E2 18929.918} C_VEL
LIN {X 0,Y 420.352,Z 384.991,A -85,B 0,C 180,E1 18929.184,E2 18929.184} C_VEL
LIN {X 0,Y 417.737,Z 380.687,A -85,B 0,C 180,E1 18927.977,E2 18927.977} C_VEL
LIN {X 0,Y 417.345,Z 379.214,A -85,B 0,C 180,E1 18927.54,E2 18927.54} C_VEL
LIN {X 0,Y 417.352,Z 379.051,A -85,B 0,C 180,E1 18923.733,E2 18923.733} C_VEL
LIN {X 0,Y 417.345,Z 379.052,A -85,B 0,C 180,E1 18919.888,E2 18919.888} C_VEL
LIN {X 0,Y 417.323,Z 379.062,A -85,B 0,C 180,E1 18916.126,E2 18916.126} C_VEL
LIN {X 0,Y 417.312,Z 379.066,A -85,B 0,C 180,E1 18912.452,E2 18912.452} C_VEL
LIN {X 0,Y 417.315,Z 379.057,A -85,B 0,C 180,E1 18908.542,E2 18908.542} C_VEL
LIN {X 0,Y 417.335,Z 379.05,A -85,B 0,C 180,E1 18904.81,E2 18904.81} C_VEL
LIN {X 0,Y 417.361,Z 379.048,A -85,B 0,C 180,E1 18900.96,E2 18900.96} C_VEL
LIN {X 0,Y 417.366,Z 379.049,A -85,B 0,C 180,E1 18897.116,E2 18897.116} C_VEL
LIN {X 0,Y 417.355,Z 379.053,A -85,B 0,C 180,E1 18893.258,E2 18893.258} C_VEL
LIN {X 0,Y 417.336,Z 379.058,A -85,B 0,C 180,E1 18889.509,E2 18889.509} C_VEL
LIN {X 0,Y 417.331,Z 379.061,A -85,B 0,C 180,E1 18885.713,E2 18885.713} C_VEL
LIN {X 0,Y 417.341,Z 379.062,A -85,B 0,C 180,E1 18881.853,E2 18881.853} C_VEL
LIN {X 0,Y 417.359,Z 379.06,A -85,B 0,C 180,E1 18878.054,E2 18878.054} C_VEL
LIN {X 0,Y 417.379,Z 379.056,A -85,B 0,C 180,E1 18874.242,E2 18874.242} C_VEL
LIN {X 0,Y 417.384,Z 379.051,A -85,B 0,C 180,E1 18870.399,E2 18870.399} C_VEL
LIN {X 0,Y 417.367,Z 379.05,A -85,B 0,C 180,E1 18866.564,E2 18866.564} C_VEL
LIN {X 0,Y 417.354,Z 379.05,A -85,B 0,C 180,E1 18862.682,E2 18862.682} C_VEL
LIN {X 0,Y 417.35,Z 379.048,A -85,B 0,C 180,E1 18858.971,E2 18858.971} C_VEL
LIN {X 0,Y 417.36,Z 379.056,A -85,B 0,C 180,E1 18855.156,E2 18855.156} C_VEL
LIN {X 0,Y 417.382,Z 379.057,A -85,B 0,C 180,E1 18851.383,E2 18851.383} C_VEL
LIN {X 0,Y 417.378,Z 379.048,A -85,B 0,C 180,E1 18847.473,E2 18847.473} C_VEL
LIN {X 0,Y 417.381,Z 379.054,A -85,B 0,C 180,E1 18843.524,E2 18843.524} C_VEL
LIN {X 0,Y 417.381,Z 379.037,A -85,B 0,C 180,E1 18839.565,E2 18839.565} C_VEL
LIN {X 0,Y 417.485,Z 379.661,A -85,B 0,C 180,E1 18839.054,E2 18839.054} C_VEL
LIN {X 0,Y 418.886,Z 382.832,A -85,B 0,C 180,E1 18838.51,E2 18838.51} C_VEL
LIN {X 0,Y 421.685,Z 385.199,A -85,B 0,C 180,E1 18837.819,E2 18837.819} C_VEL
LIN {X 0,Y 422.433,Z 386.12,A -85,B 0,C 180,E1 18837.625,E2 18837.625} C_VEL
LIN {X 0,Y 424.872,Z 389.776,A -85,B 0,C 180,E1 18836.976,E2 18836.976} C_VEL
LIN {X 0,Y 427.194,Z 392.011,A -85,B 0,C 180,E1 18836.415,E2 18836.415} C_VEL
LIN {X 0,Y 430.334,Z 396.198,A -85,B 0,C 180,E1 18835.643,E2 18835.643} C_VEL
LIN {X 0,Y 431.988,Z 398.149,A -85,B 0,C 180,E1 18835.255,E2 18835.255} C_VEL
LIN {X 0,Y 435.669,Z 402.626,A -85,B 0,C 180,E1 18834.411,E2 18834.411} C_VEL
LIN {X 0,Y 448.329,Z 419.098,A -85,B 0,C 180,E1 18831.688,E2 18831.688} C_VEL
LIN {X 0,Y 459.668,Z 434.793,A -85,B 0,C 180,E1 18829.448,E2 18829.448} C_VEL
LIN {X 0,Y 466.284,Z 444.453,A -85,B 0,C 180,E1 18828.222,E2 18828.222} C_VEL
LIN {X 0,Y 462.784,Z 536.379,A -85,B 0,C 180,E1 18826.537,E2 18826.537} C_VEL
LIN {X 0,Y 461.86,Z 544.077,A -85,B 0,C 180,E1 18826.485,E2 18826.485} C_VEL
LIN {X 0,Y 456.883,Z 564.679,A -85,B 0,C 180,E1 18826.693,E2 18826.693} C_VEL
LIN {X 0,Y 456.139,Z 571.285,A -85,B 0,C 180,E1 18826.641,E2 18826.641} C_VEL
LIN {X 0,Y 450.757,Z 713.595,A -85,B 0,C 180,E1 18824.02,E2 18824.02} C_VEL
LIN {X 0,Y 448.971,Z 736.809,A -85,B 0,C 180,E1 18823.4,E2 18823.4} C_VEL
LIN {X 0,Y 446.787,Z 758.889,A -85,B 0,C 180,E1 18822.599,E2 18822.599} C_VEL
LIN {X 0,Y 444.132,Z 779.624,A -85,B 0,C 180,E1 18821.62,E2 18821.62} C_VEL
LIN {X 0,Y 441.151,Z 800.148,A -85,B 0,C 180,E1 18820.443,E2 18820.443} C_VEL
LIN {X 0,Y 437.647,Z 820.697,A -85,B 0,C 180,E1 18819,E2 18819} C_VEL
LIN {X 0,Y 433.989,Z 840.629,A -85,B 0,C 180,E1 18817.342,E2 18817.342} C_VEL
LIN {X 0,Y 430.324,Z 858.95,A -85,B 0,C 180,E1 18815.53,E2 18815.53} C_VEL
LIN {X 0,Y 426.413,Z 877.751,A -85,B 0,C 180,E1 18813.357,E2 18813.357} C_VEL
LIN {X 0,Y 423.005,Z 893.615,A -85,B 0,C 180,E1 18811.215,E2 18811.215} C_VEL
LIN {X 0,Y 419.492,Z 910.049,A -85,B 0,C 180,E1 18808.631,E2 18808.631} C_VEL
LIN {X 0,Y 416.522,Z 924.436,A -85,B 0,C 180,E1 18806.005,E2 18806.005} C_VEL
LIN {X 0,Y 413.817,Z 938.079,A -85,B 0,C 180,E1 18803.058,E2 18803.058} C_VEL
LIN {X 0,Y 411.635,Z 950.362,A -85,B 0,C 180,E1 18799.925,E2 18799.925} C_VEL
LIN {X 0,Y 410.115,Z 960.35,A -85,B 0,C 180,E1 18796.892,E2 18796.892} C_VEL
LIN {X 0,Y 409.023,Z 969.047,A -85,B 0,C 180,E1 18793.67,E2 18793.67} C_VEL
LIN {X 0,Y 408.382,Z 975.906,A -85,B 0,C 180,E1 18790.496,E2 18790.496} C_VEL
LIN {X 0,Y 408.057,Z 981.356,A -85,B 0,C 180,E1 18787.22,E2 18787.22} C_VEL
LIN {X 0,Y 407.922,Z 985.04,A -85,B 0,C 180,E1 18784.101,E2 18784.101} C_VEL
LIN {X 0,Y 407.92,Z 987.257,A -85,B 0,C 180,E1 18780.963,E2 18780.963} C_VEL
LIN {X 0,Y 407.905,Z 987.992,A -85,B 0,C 180,E1 18777.862,E2 18777.862} C_VEL
LIN {X 0,Y 407.913,Z 987.162,A -85,B 0,C 180,E1 18774.71,E2 18774.71} C_VEL
LIN {X 0,Y 407.931,Z 984.9,A -85,B 0,C 180,E1 18771.66,E2 18771.66} C_VEL
LIN {X 0,Y 408.072,Z 981.174,A -85,B 0,C 180,E1 18768.57,E2 18768.57} C_VEL
LIN {X 0,Y 408.39,Z 975.797,A -85,B 0,C 180,E1 18765.356,E2 18765.356} C_VEL
LIN {X 0,Y 409.035,Z 969.001,A -85,B 0,C 180,E1 18762.209,E2 18762.209} C_VEL
LIN {X 0,Y 410.152,Z 960.206,A -85,B 0,C 180,E1 18758.951,E2 18758.951} C_VEL
LIN {X 0,Y 411.756,Z 949.873,A -85,B 0,C 180,E1 18755.819,E2 18755.819} C_VEL
LIN {X 0,Y 413.916,Z 937.8,A -85,B 0,C 180,E1 18752.759,E2 18752.759} C_VEL
LIN {X 0,Y 416.529,Z 924.755,A -85,B 0,C 180,E1 18749.935,E2 18749.935} C_VEL
LIN {X 0,Y 419.387,Z 910.942,A -85,B 0,C 180,E1 18747.396,E2 18747.396} C_VEL
LIN {X 0,Y 422.926,Z 894.512,A -85,B 0,C 180,E1 18744.789,E2 18744.789} C_VEL
LIN {X 0,Y 426.359,Z 878.542,A -85,B 0,C 180,E1 18742.619,E2 18742.619} C_VEL
LIN {X 0,Y 430.183,Z 860.306,A -85,B 0,C 180,E1 18740.495,E2 18740.495} C_VEL
LIN {X 0,Y 433.815,Z 842.198,A -85,B 0,C 180,E1 18738.684,E2 18738.684} C_VEL
LIN {X 0,Y 437.499,Z 822.329,A -85,B 0,C 180,E1 18737.01,E2 18737.01} C_VEL
LIN {X 0,Y 441.063,Z 801.565,A -85,B 0,C 180,E1 18735.534,E2 18735.534} C_VEL
LIN {X 0,Y 444.082,Z 780.941,A -85,B 0,C 180,E1 18734.34,E2 18734.34} C_VEL
LIN {X 0,Y 446.826,Z 759.501,A -85,B 0,C 180,E1 18733.321,E2 18733.321} C_VEL
LIN {X 0,Y 449.036,Z 737.238,A -85,B 0,C 180,E1 18732.511,E2 18732.511} C_VEL
LIN {X 0,Y 450.829,Z 713.469,A -85,B 0,C 180,E1 18731.879,E2 18731.879} C_VEL
LIN {X 0,Y 459.541,Z 500.737,A -85,B 0,C 180,E1 18727.899,E2 18727.899} C_VEL
LIN {X 0,Y 461.818,Z 448.371,A -85,B 0,C 180,E1 18726.886,E2 18726.886} C_VEL
LIN {X 0,Y 452.246,Z 434.182,A -85,B 0,C 180,E1 18724.82,E2 18724.82} C_VEL
LIN {X 0,Y 445.006,Z 424.146,A -85,B 0,C 180,E1 18723.092,E2 18723.092} C_VEL
LIN {X 0,Y 438.877,Z 415.887,A -85,B 0,C 180,E1 18721.469,E2 18721.469} C_VEL
LIN {X 0,Y 434.5,Z 410.338,A -85,B 0,C 180,E1 18720.198,E2 18720.198} C_VEL
LIN {X 0,Y 430.484,Z 405.207,A -85,B 0,C 180,E1 18718.936,E2 18718.936} C_VEL
LIN {X 0,Y 427.259,Z 401.516,A -85,B 0,C 180,E1 18717.822,E2 18717.822} C_VEL
LIN {X 0,Y 426.111,Z 399.584,A -85,B 0,C 180,E1 18717.378,E2 18717.378} C_VEL
LIN {X 0,Y 422.891,Z 396.744,A -85,B 0,C 180,E1 18716.179,E2 18716.179} C_VEL
LIN {X 0,Y 421.028,Z 393.41,A -85,B 0,C 180,E1 18715.301,E2 18715.301} C_VEL
LIN {X 0,Y 417.562,Z 390.874,A -85,B 0,C 180,E1 18713.746,E2 18713.746} C_VEL
LIN {X 0,Y 415.79,Z 387.639,A -85,B 0,C 180,E1 18712.643,E2 18712.643} C_VEL
LIN {X 0,Y 414.639,Z 386.602,A -85,B 0,C 180,E1 18711.961,E2 18711.961} C_VEL
LIN {X 0,Y 410.933,Z 383.833,A -85,B 0,C 180,E1 18709.202,E2 18709.202} C_VEL
LIN {X 0,Y 409.566,Z 380.885,A -85,B 0,C 180,E1 18706.93,E2 18706.93} C_VEL
LIN {X 0,Y 409.471,Z 380.256,A -85,B 0,C 180,E1 18704.129,E2 18704.129} C_VEL
LIN {X 0,Y 409.564,Z 380.904,A -85,B 0,C 180,E1 18701.497,E2 18701.497} C_VEL
LIN {X 0,Y 410.699,Z 383.511,A -85,B 0,C 180,E1 18699.478,E2 18699.478} C_VEL
LIN {X 0,Y 414.279,Z 386.46,A -85,B 0,C 180,E1 18696.684,E2 18696.684} C_VEL
LIN {X 0,Y 415.681,Z 387.433,A -85,B 0,C 180,E1 18695.864,E2 18695.864} C_VEL
LIN {X 0,Y 417.424,Z 390.74,A -85,B 0,C 180,E1 18694.763,E2 18694.763} C_VEL
LIN {X 0,Y 420.911,Z 393.876,A -85,B 0,C 180,E1 18693.133,E2 18693.133} C_VEL
LIN {X 0,Y 424.572,Z 398.589,A -85,B 0,C 180,E1 18691.595,E2 18691.595} C_VEL
LIN {X 0,Y 429.505,Z 404.939,A -85,B 0,C 180,E1 18689.813,E2 18689.813} C_VEL
LIN {X 0,Y 434.181,Z 411.388,A -85,B 0,C 180,E1 18688.29,E2 18688.29} C_VEL
LIN {X 0,Y 440.741,Z 420.665,A -85,B 0,C 180,E1 18686.391,E2 18686.391} C_VEL
LIN {X 0,Y 448.811,Z 432.761,A -85,B 0,C 180,E1 18684.33,E2 18684.33} C_VEL
LIN {X 0,Y 458.037,Z 447.62,A -85,B 0,C 180,E1 18682.224,E2 18682.224} C_VEL
LIN {X 0,Y 461.89,Z 454.532,A -85,B 0,C 180,E1 18681.397,E2 18681.397} C_VEL
LIN {X 0,Y 453.826,Z 646.988,A -85,B 0,C 180,E1 18677.778,E2 18677.778} C_VEL
LIN {X 0,Y 450.271,Z 737.997,A -85,B 0,C 180,E1 18676.079,E2 18676.079} C_VEL
LIN {X 0,Y 448.275,Z 761.497,A -85,B 0,C 180,E1 18675.452,E2 18675.452} C_VEL
LIN {X 0,Y 445.858,Z 784.221,A -85,B 0,C 180,E1 18674.629,E2 18674.629} C_VEL
LIN {X 0,Y 443.069,Z 805.393,A -85,B 0,C 180,E1 18673.631,E2 18673.631} C_VEL
LIN {X 0,Y 439.684,Z 828.043,A -85,B 0,C 180,E1 18672.311,E2 18672.311} C_VEL
LIN {X 0,Y 436.405,Z 847.459,A -85,B 0,C 180,E1 18670.942,E2 18670.942} C_VEL
LIN {X 0,Y 432.472,Z 868.953,A -85,B 0,C 180,E1 18669.139,E2 18669.139} C_VEL
LIN {X 0,Y 428.803,Z 888.137,A -85,B 0,C 180,E1 18667.238,E2 18667.238} C_VEL
LIN {X 0,Y 425.236,Z 905.849,A -85,B 0,C 180,E1 18665.177,E2 18665.177} C_VEL
LIN {X 0,Y 421.8,Z 923.045,A -85,B 0,C 180,E1 18662.88,E2 18662.88} C_VEL
LIN {X 0,Y 418.649,Z 938.723,A -85,B 0,C 180,E1 18660.422,E2 18660.422} C_VEL
LIN {X 0,Y 415.741,Z 954.031,A -85,B 0,C 180,E1 18657.659,E2 18657.659} C_VEL
LIN {X 0,Y 413.494,Z 966.471,A -85,B 0,C 180,E1 18655.037,E2 18655.037} C_VEL
LIN {X 0,Y 411.482,Z 978.956,A -85,B 0,C 180,E1 18651.978,E2 18651.978} C_VEL
LIN {X 0,Y 410.145,Z 988.494,A -85,B 0,C 180,E1 18649.218,E2 18649.218} C_VEL
LIN {X 0,Y 409.049,Z 998.074,A -85,B 0,C 180,E1 18645.892,E2 18645.892} C_VEL
LIN {X 0,Y 408.456,Z 1004.79,A -85,B 0,C 180,E1 18643.018,E2 18643.018} C_VEL
LIN {X 0,Y 408.082,Z 1010.424,A -85,B 0,C 180,E1 18639.879,E2 18639.879} C_VEL
LIN {X 0,Y 407.939,Z 1013.955,A -85,B 0,C 180,E1 18637.184,E2 18637.184} C_VEL
LIN {X 0,Y 407.911,Z 1016.71,A -85,B 0,C 180,E1 18634.08,E2 18634.08} C_VEL
LIN {X 0,Y 407.898,Z 1017.825,A -85,B 0,C 180,E1 18631.127,E2 18631.127} C_VEL
LIN {X 0,Y 407.906,Z 1017.735,A -85,B 0,C 180,E1 18628.318,E2 18628.318} C_VEL
LIN {X 0,Y 407.913,Z 1016.07,A -85,B 0,C 180,E1 18625.082,E2 18625.082} C_VEL
LIN {X 0,Y 407.962,Z 1013.483,A -85,B 0,C 180,E1 18622.399,E2 18622.399} C_VEL
LIN {X 0,Y 408.176,Z 1008.963,A -85,B 0,C 180,E1 18619.195,E2 18619.195} C_VEL
LIN {X 0,Y 408.547,Z 1003.566,A -85,B 0,C 180,E1 18616.416,E2 18616.416} C_VEL
LIN {X 0,Y 409.278,Z 995.886,A -85,B 0,C 180,E1 18613.25,E2 18613.25} C_VEL
LIN {X 0,Y 410.325,Z 987.187,A -85,B 0,C 180,E1 18610.355,E2 18610.355} C_VEL
LIN {X 0,Y 411.937,Z 976.255,A -85,B 0,C 180,E1 18607.269,E2 18607.269} C_VEL
LIN {X 0,Y 413.851,Z 964.767,A -85,B 0,C 180,E1 18604.535,E2 18604.535} C_VEL
LIN {X 0,Y 416.469,Z 950.577,A -85,B 0,C 180,E1 18601.623,E2 18601.623} C_VEL
LIN {X 0,Y 419.228,Z 936.594,A -85,B 0,C 180,E1 18599.157,E2 18599.157} C_VEL
LIN {X 0,Y 422.682,Z 919.531,A -85,B 0,C 180,E1 18596.559,E2 18596.559} C_VEL
LIN {X 0,Y 426.177,Z 902.66,A -85,B 0,C 180,E1 18594.343,E2 18594.343} C_VEL
LIN {X 0,Y 429.862,Z 884.114,A -85,B 0,C 180,E1 18592.263,E2 18592.263} C_VEL
LIN {X 0,Y 433.675,Z 864.702,A -85,B 0,C 180,E1 18590.393,E2 18590.393} C_VEL
LIN {X 0,Y 437.219,Z 844.957,A -85,B 0,C 180,E1 18588.796,E2 18588.796} C_VEL
LIN {X 0,Y 440.679,Z 824.244,A -85,B 0,C 180,E1 18587.376,E2 18587.376} C_VEL
LIN {X 0,Y 443.654,Z 803.821,A -85,B 0,C 180,E1 18586.227,E2 18586.227} C_VEL
LIN {X 0,Y 446.609,Z 780.553,A -85,B 0,C 180,E1 18585.176,E2 18585.176} C_VEL
LIN {X 0,Y 448.8,Z 759.176,A -85,B 0,C 180,E1 18584.438,E2 18584.438} C_VEL
LIN {X 0,Y 450.637,Z 734.595,A -85,B 0,C 180,E1 18583.827,E2 18583.827} C_VEL
LIN {X 0,Y 458.506,Z 524.422,A -85,B 0,C 180,E1 18579.963,E2 18579.963} C_VEL
LIN {X 0,Y 461.166,Z 454.19,A -85,B 0,C 180,E1 18578.639,E2 18578.639} C_VEL
LIN {X 0,Y 449.037,Z 435.384,A -85,B 0,C 180,E1 18576.24,E2 18576.24} C_VEL
LIN {X 0,Y 436.459,Z 417.213,A -85,B 0,C 180,E1 18573.51,E2 18573.51} C_VEL
LIN {X 0,Y 427.73,Z 405.58,A -85,B 0,C 180,E1 18571.457,E2 18571.457} C_VEL
LIN {X 0,Y 420.324,Z 395.803,A -85,B 0,C 180,E1 18569.577,E2 18569.577} C_VEL
LIN {X 0,Y 416.125,Z 390.454,A -85,B 0,C 180,E1 18568.447,E2 18568.447} C_VEL
LIN {X 0,Y 413.035,Z 386.491,A -85,B 0,C 180,E1 18567.578,E2 18567.578} C_VEL
LIN {X 0,Y 411.666,Z 384.758,A -85,B 0,C 180,E1 18567.168,E2 18567.168} C_VEL
LIN {X 0,Y 409.713,Z 381.506,A -85,B 0,C 180,E1 18566.212,E2 18566.212} C_VEL
LIN {X 0,Y 409.426,Z 380.186,A -85,B 0,C 180,E1 18565.765,E2 18565.765} C_VEL
LIN {X 0,Y 409.424,Z 380.047,A -85,B 0,C 180,E1 18561.789,E2 18561.789} C_VEL
LIN {X 0,Y 409.412,Z 380.041,A -85,B 0,C 180,E1 18557.758,E2 18557.758} C_VEL
LIN {X 0,Y 409.39,Z 380.041,A -85,B 0,C 180,E1 18553.992,E2 18553.992} C_VEL
LIN {X 0,Y 409.378,Z 380.048,A -85,B 0,C 180,E1 18550.204,E2 18550.204} C_VEL
LIN {X 0,Y 409.378,Z 380.054,A -85,B 0,C 180,E1 18546.306,E2 18546.306} C_VEL
LIN {X 0,Y 409.383,Z 380.052,A -85,B 0,C 180,E1 18542.379,E2 18542.379} C_VEL
LIN {X 0,Y 409.4,Z 380.045,A -85,B 0,C 180,E1 18538.6,E2 18538.6} C_VEL
LIN {X 0,Y 409.426,Z 380.036,A -85,B 0,C 180,E1 18534.815,E2 18534.815} C_VEL
LIN {X 0,Y 409.431,Z 380.036,A -85,B 0,C 180,E1 18531.008,E2 18531.008} C_VEL
LIN {X 0,Y 409.414,Z 380.037,A -85,B 0,C 180,E1 18527.159,E2 18527.159} C_VEL
LIN {X 0,Y 409.399,Z 380.038,A -85,B 0,C 180,E1 18523.396,E2 18523.396} C_VEL
LIN {X 0,Y 409.399,Z 380.038,A -85,B 0,C 180,E1 18519.559,E2 18519.559} C_VEL
LIN {X 0,Y 409.407,Z 380.04,A -85,B 0,C 180,E1 18515.776,E2 18515.776} C_VEL
LIN {X 0,Y 409.436,Z 380.039,A -85,B 0,C 180,E1 18512.038,E2 18512.038} C_VEL
LIN {X 0,Y 409.446,Z 380.042,A -85,B 0,C 180,E1 18508.165,E2 18508.165} C_VEL
LIN {X 0,Y 409.438,Z 380.049,A -85,B 0,C 180,E1 18504.292,E2 18504.292} C_VEL
LIN {X 0,Y 409.43,Z 380.044,A -85,B 0,C 180,E1 18500.403,E2 18500.403} C_VEL
LIN {X 0,Y 409.415,Z 380.041,A -85,B 0,C 180,E1 18496.666,E2 18496.666} C_VEL
LIN {X 0,Y 409.414,Z 380.038,A -85,B 0,C 180,E1 18492.753,E2 18492.753} C_VEL
LIN {X 0,Y 409.422,Z 380.049,A -85,B 0,C 180,E1 18488.827,E2 18488.827} C_VEL
LIN {X 0,Y 409.425,Z 380.04,A -85,B 0,C 180,E1 18484.86,E2 18484.86} C_VEL
LIN {X 0,Y 409.474,Z 380.251,A -85,B 0,C 180,E1 18481.088,E2 18481.088} C_VEL
LIN {X 0,Y 409.838,Z 381.73,A -85,B 0,C 180,E1 18480.686,E2 18480.686} C_VEL
LIN {X 0,Y 411.722,Z 384.688,A -85,B 0,C 180,E1 18480.1,E2 18480.1} C_VEL
LIN {X 0,Y 414.406,Z 386.844,A -85,B 0,C 180,E1 18479.389,E2 18479.389} C_VEL
LIN {X 0,Y 416.741,Z 390.557,A -85,B 0,C 180,E1 18478.726,E2 18478.726} C_VEL
LIN {X 0,Y 419.476,Z 393.094,A -85,B 0,C 180,E1 18478.035,E2 18478.035} C_VEL
LIN {X 0,Y 422.541,Z 397.218,A -85,B 0,C 180,E1 18477.234,E2 18477.234} C_VEL
LIN {X 0,Y 424.352,Z 399.134,A -85,B 0,C 180,E1 18476.784,E2 18476.784} C_VEL
LIN {X 0,Y 427.928,Z 403.603,A -85,B 0,C 180,E1 18475.899,E2 18475.899} C_VEL
LIN {X 0,Y 438.547,Z 417.315,A -85,B 0,C 180,E1 18473.452,E2 18473.452} C_VEL
LIN {X 0,Y 449.217,Z 431.538,A -85,B 0,C 180,E1 18471.204,E2 18471.204} C_VEL
LIN {X 0,Y 460.984,Z 448.291,A -85,B 0,C 180,E1 18468.913,E2 18468.913} C_VEL
LIN {X 0,Y 456.139,Z 571.285,A -85,B 0,C 180,E1 18466.641,E2 18466.641} C_VEL
LIN {X 0,Y 455.187,Z 578.983,A -85,B 0,C 180,E1 18466.591,E2 18466.591} C_VEL
LIN {X 0,Y 450.167,Z 599.57,A -85,B 0,C 180,E1 18466.806,E2 18466.806} C_VEL
LIN {X 0,Y 449.416,Z 606.174,A -85,B 0,C 180,E1 18466.753,E2 18466.753} C_VEL
LIN {X 0,Y 445.113,Z 714.172,A -85,B 0,C 180,E1 18464.742,E2 18464.742} C_VEL
LIN {X 0,Y 443.247,Z 737.29,A -85,B 0,C 180,E1 18464.117,E2 18464.117} C_VEL
LIN {X 0,Y 440.943,Z 759.529,A -85,B 0,C 180,E1 18463.302,E2 18463.302} C_VEL
LIN {X 0,Y 438.175,Z 780.223,A -85,B 0,C 180,E1 18462.315,E2 18462.315} C_VEL
LIN {X 0,Y 434.906,Z 801.693,A -85,B 0,C 180,E1 18461.065,E2 18461.065} C_VEL
LIN {X 0,Y 431.413,Z 821.292,A -85,B 0,C 180,E1 18459.669,E2 18459.669} C_VEL
LIN {X 0,Y 427.569,Z 841.197,A -85,B 0,C 180,E1 18457.994,E2 18457.994} C_VEL
LIN {X 0,Y 423.719,Z 859.518,A -85,B 0,C 180,E1 18456.16,E2 18456.16} C_VEL
LIN {X 0,Y 419.52,Z 878.695,A -85,B 0,C 180,E1 18453.907,E2 18453.907} C_VEL
LIN {X 0,Y 416.022,Z 894.165,A -85,B 0,C 180,E1 18451.787,E2 18451.787} C_VEL
LIN {X 0,Y 412.307,Z 910.565,A -85,B 0,C 180,E1 18449.163,E2 18449.163} C_VEL
LIN {X 0,Y 409.153,Z 924.936,A -85,B 0,C 180,E1 18446.494,E2 18446.494} C_VEL
LIN {X 0,Y 406.404,Z 937.924,A -85,B 0,C 180,E1 18443.64,E2 18443.64} C_VEL
LIN {X 0,Y 404.151,Z 949.792,A -85,B 0,C 180,E1 18440.599,E2 18440.599} C_VEL
LIN {X 0,Y 402.456,Z 959.861,A -85,B 0,C 180,E1 18437.514,E2 18437.514} C_VEL
LIN {X 0,Y 401.199,Z 968.909,A -85,B 0,C 180,E1 18434.151,E2 18434.151} C_VEL
LIN {X 0,Y 400.49,Z 975.575,A -85,B 0,C 180,E1 18431.058,E2 18431.058} C_VEL
LIN {X 0,Y 400.113,Z 980.955,A -85,B 0,C 180,E1 18427.828,E2 18427.828} C_VEL
LIN {X 0,Y 399.947,Z 984.908,A -85,B 0,C 180,E1 18424.489,E2 18424.489} C_VEL
LIN {X 0,Y 399.918,Z 987.188,A -85,B 0,C 180,E1 18421.309,E2 18421.309} C_VEL
LIN {X 0,Y 399.905,Z 988.02,A -85,B 0,C 180,E1 18417.988,E2 18417.988} C_VEL
LIN {X 0,Y 399.913,Z 987.237,A -85,B 0,C 180,E1 18414.719,E2 18414.719} C_VEL
LIN {X 0,Y 399.947,Z 984.979,A -85,B 0,C 180,E1 18411.49,E2 18411.49} C_VEL
LIN {X 0,Y 400.108,Z 981.336,A -85,B 0,C 180,E1 18408.336,E2 18408.336} C_VEL
LIN {X 0,Y 400.465,Z 975.983,A -85,B 0,C 180,E1 18405.04,E2 18405.04} C_VEL
LIN {X 0,Y 401.162,Z 969.327,A -85,B 0,C 180,E1 18401.911,E2 18401.911} C_VEL
LIN {X 0,Y 402.379,Z 960.536,A -85,B 0,C 180,E1 18398.588,E2 18398.588} C_VEL
LIN {X 0,Y 404.046,Z 950.554,A -85,B 0,C 180,E1 18395.493,E2 18395.493} C_VEL
LIN {X 0,Y 406.303,Z 938.747,A -85,B 0,C 180,E1 18392.423,E2 18392.423} C_VEL
LIN {X 0,Y 409.085,Z 925.697,A -85,B 0,C 180,E1 18389.525,E2 18389.525} C_VEL
LIN {X 0,Y 412.28,Z 911.19,A -85,B 0,C 180,E1 18386.811,E2 18386.811} C_VEL
LIN {X 0,Y 415.982,Z 894.942,A -85,B 0,C 180,E1 18384.194,E2 18384.194} C_VEL
LIN {X 0,Y 419.667,Z 878.749,A -85,B 0,C 180,E1 18381.966,E2 18381.966} C_VEL
LIN {X 0,Y 423.845,Z 859.747,A -85,B 0,C 180,E1 18379.733,E2 18379.733} C_VEL
LIN {X 0,Y 427.886,Z 840.676,A -85,B 0,C 180,E1 18377.826,E2 18377.826} C_VEL
LIN {X 0,Y 431.603,Z 821.362,A -85,B 0,C 180,E1 18376.21,E2 18376.21} C_VEL
LIN {X 0,Y 435.284,Z 800.639,A -85,B 0,C 180,E1 18374.744,E2 18374.744} C_VEL
LIN {X 0,Y 438.321,Z 780.734,A -85,B 0,C 180,E1 18373.589,E2 18373.589} C_VEL
LIN {X 0,Y 441.204,Z 758.975,A -85,B 0,C 180,E1 18372.556,E2 18372.556} C_VEL
LIN {X 0,Y 443.482,Z 737.059,A -85,B 0,C 180,E1 18371.758,E2 18371.758} C_VEL
LIN {X 0,Y 445.393,Z 712.189,A -85,B 0,C 180,E1 18371.106,E2 18371.106} C_VEL
LIN {X 0,Y 454.557,Z 501.455,A -85,B 0,C 180,E1 18367.119,E2 18367.119} C_VEL
LIN {X 0,Y 456.792,Z 452.505,A -85,B 0,C 180,E1 18366.157,E2 18366.157} C_VEL
LIN {X 0,Y 448.076,Z 439.372,A -85,B 0,C 180,E1 18364.184,E2 18364.184} C_VEL
LIN {X 0,Y 440.032,Z 427.986,A -85,B 0,C 180,E1 18362.149,E2 18362.149} C_VEL
LIN {X 0,Y 435.143,Z 421.644,A -85,B 0,C 180,E1 18360.79,E2 18360.79} C_VEL
LIN {X 0,Y 431.952,Z 417.387,A -85,B 0,C 180,E1 18359.818,E2 18359.818} C_VEL
LIN {X 0,Y 427.996,Z 412.316,A -85,B 0,C 180,E1 18358.528,E2 18358.528} C_VEL
LIN {X 0,Y 424.694,Z 408.194,A -85,B 0,C 180,E1 18357.335,E2 18357.335} C_VEL
LIN {X 0,Y 423.703,Z 406.854,A -85,B 0,C 180,E1 18356.957,E2 18356.957} C_VEL
LIN {X 0,Y 420.517,Z 403.527,A -85,B 0,C 180,E1 18355.671,E2 18355.671} C_VEL
LIN {X 0,Y 418.981,Z 400.934,A -85,B 0,C 180,E1 18354.935,E2 18354.935} C_VEL
LIN {X 0,Y 415.716,Z 398.207,A -85,B 0,C 180,E1 18353.371,E2 18353.371} C_VEL
LIN {X 0,Y 413.704,Z 394.652,A -85,B 0,C 180,E1 18352.082,E2 18352.082} C_VEL
LIN {X 0,Y 409.908,Z 391.986,A -85,B 0,C 180,E1 18349.317,E2 18349.317} C_VEL
LIN {X 0,Y 408.066,Z 388.565,A -85,B 0,C 180,E1 18346.6,E2 18346.6} C_VEL
LIN {X 0,Y 407.537,Z 388.068,A -85,B 0,C 180,E1 18343.6,E2 18343.6} C_VEL
LIN {X 0,Y 408.248,Z 388.883,A -85,B 0,C 180,E1 18341.415,E2 18341.415} C_VEL
LIN {X 0,Y 410.994,Z 393.066,A -85,B 0,C 180,E1 18338.148,E2 18338.148} C_VEL
LIN {X 0,Y 413.991,Z 395.006,A -85,B 0,C 180,E1 18336.176,E2 18336.176} C_VEL
LIN {X 0,Y 415.879,Z 398.463,A -85,B 0,C 180,E1 18334.968,E2 18334.968} C_VEL
LIN {X 0,Y 419.135,Z 401.496,A -85,B 0,C 180,E1 18333.393,E2 18333.393} C_VEL
LIN {X 0,Y 422.717,Z 406.149,A -85,B 0,C 180,E1 18331.844,E2 18331.844} C_VEL
LIN {X 0,Y 427.358,Z 412.431,A -85,B 0,C 180,E1 18330.11,E2 18330.11} C_VEL
LIN {X 0,Y 431.735,Z 418.578,A -85,B 0,C 180,E1 18328.635,E2 18328.635} C_VEL
LIN {X 0,Y 438.187,Z 427.909,A -85,B 0,C 180,E1 18326.718,E2 18326.718} C_VEL
LIN {X 0,Y 445.636,Z 439.351,A -85,B 0,C 180,E1 18324.752,E2 18324.752} C_VEL
LIN {X 0,Y 454.389,Z 453.746,A -85,B 0,C 180,E1 18322.684,E2 18322.684} C_VEL
LIN {X 0,Y 456.876,Z 458.487,A -85,B 0,C 180,E1 18322.123,E2 18322.123} C_VEL
LIN {X 0,Y 448.41,Z 648.672,A -85,B 0,C 180,E1 18318.507,E2 18318.507} C_VEL
LIN {X 0,Y 444.674,Z 738.199,A -85,B 0,C 180,E1 18316.812,E2 18316.812} C_VEL
LIN {X 0,Y 442.574,Z 761.654,A -85,B 0,C 180,E1 18316.178,E2 18316.178} C_VEL
LIN {X 0,Y 439.998,Z 784.446,A -85,B 0,C 180,E1 18315.341,E2 18315.341} C_VEL
LIN {X 0,Y 437.081,Z 805.486,A -85,B 0,C 180,E1 18314.338,E2 18314.338} C_VEL
LIN {X 0,Y 433.465,Z 828.437,A -85,B 0,C 180,E1 18312.982,E2 18312.982} C_VEL
LIN {X 0,Y 430.186,Z 846.929,A -85,B 0,C 180,E1 18311.665,E2 18311.665} C_VEL
LIN {X 0,Y 426.046,Z 868.43,A -85,B 0,C 180,E1 18309.846,E2 18309.846} C_VEL
LIN {X 0,Y 422.192,Z 887.468,A -85,B 0,C 180,E1 18307.943,E2 18307.943} C_VEL
LIN {X 0,Y 418.405,Z 905.351,A -85,B 0,C 180,E1 18305.839,E2 18305.839} C_VEL
LIN {X 0,Y 414.756,Z 922.569,A -85,B 0,C 180,E1 18303.511,E2 18303.511} C_VEL
LIN {X 0,Y 411.416,Z 938.27,A -85,B 0,C 180,E1 18301.015,E2 18301.015} C_VEL
LIN {X 0,Y 408.448,Z 952.882,A -85,B 0,C 180,E1 18298.356,E2 18298.356} C_VEL
LIN {X 0,Y 405.911,Z 966.063,A -85,B 0,C 180,E1 18295.538,E2 18295.538} C_VEL
LIN {X 0,Y 403.757,Z 978.567,A -85,B 0,C 180,E1 18292.421,E2 18292.421} C_VEL
LIN {X 0,Y 402.315,Z 988.122,A -85,B 0,C 180,E1 18289.607,E2 18289.607} C_VEL
LIN {X 0,Y 401.135,Z 997.72,A -85,B 0,C 180,E1 18286.214,E2 18286.214} C_VEL
LIN {X 0,Y 400.498,Z 1004.447,A -85,B 0,C 180,E1 18283.282,E2 18283.282} C_VEL
LIN {X 0,Y 400.085,Z 1010.413,A -85,B 0,C 180,E1 18279.933,E2 18279.933} C_VEL
LIN {X 0,Y 399.939,Z 1014.007,A -85,B 0,C 180,E1 18277.184,E2 18277.184} C_VEL
LIN {X 0,Y 399.91,Z 1016.767,A -85,B 0,C 180,E1 18273.993,E2 18273.993} C_VEL
LIN {X 0,Y 399.899,Z 1017.824,A -85,B 0,C 180,E1 18271.15,E2 18271.15} C_VEL
LIN {X 0,Y 399.906,Z 1017.733,A -85,B 0,C 180,E1 18268.285,E2 18268.285} C_VEL
LIN {X 0,Y 399.912,Z 1016.144,A -85,B 0,C 180,E1 18265.128,E2 18265.128} C_VEL
LIN {X 0,Y 399.962,Z 1013.528,A -85,B 0,C 180,E1 18262.39,E2 18262.39} C_VEL
LIN {X 0,Y 400.159,Z 1009.371,A -85,B 0,C 180,E1 18259.349,E2 18259.349} C_VEL
LIN {X 0,Y 400.568,Z 1003.569,A -85,B 0,C 180,E1 18256.287,E2 18256.287} C_VEL
LIN {X 0,Y 401.297,Z 996.355,A -85,B 0,C 180,E1 18253.205,E2 18253.205} C_VEL
LIN {X 0,Y 402.442,Z 987.334,A -85,B 0,C 180,E1 18250.105,E2 18250.105} C_VEL
LIN {X 0,Y 404.13,Z 976.639,A -85,B 0,C 180,E1 18246.994,E2 18246.994} C_VEL
LIN {X 0,Y 406.297,Z 964.425,A -85,B 0,C 180,E1 18244.026,E2 18244.026} C_VEL
LIN {X 0,Y 409.132,Z 950.054,A -85,B 0,C 180,E1 18241.032,E2 18241.032} C_VEL
LIN {X 0,Y 412.025,Z 936.228,A -85,B 0,C 180,E1 18238.557,E2 18238.557} C_VEL
LIN {X 0,Y 415.708,Z 919.149,A -85,B 0,C 180,E1 18235.922,E2 18235.922} C_VEL
LIN {X 0,Y 419.357,Z 902.402,A -85,B 0,C 180,E1 18233.695,E2 18233.695} C_VEL
LIN {X 0,Y 423.246,Z 883.888,A -85,B 0,C 180,E1 18231.595,E2 18231.595} C_VEL
LIN {X 0,Y 427.277,Z 864.385,A -85,B 0,C 180,E1 18229.697,E2 18229.697} C_VEL
LIN {X 0,Y 430.997,Z 844.626,A -85,B 0,C 180,E1 18228.084,E2 18228.084} C_VEL
LIN {X 0,Y 434.688,Z 823.361,A -85,B 0,C 180,E1 18226.623,E2 18226.623} C_VEL
LIN {X 0,Y 437.765,Z 803.137,A -85,B 0,C 180,E1 18225.484,E2 18225.484} C_VEL
LIN {X 0,Y 440.951,Z 778.974,A -85,B 0,C 180,E1 18224.401,E2 18224.401} C_VEL
LIN {X 0,Y 443.192,Z 757.949,A -85,B 0,C 180,E1 18223.679,E2 18223.679} C_VEL
LIN {X 0,Y 445.022,Z 733.814,A -85,B 0,C 180,E1 18223.083,E2 18223.083} C_VEL
LIN {X 0,Y 453.219,Z 525.42,A -85,B 0,C 180,E1 18219.218,E2 18219.218} C_VEL
LIN {X 0,Y 455.941,Z 458.088,A -85,B 0,C 180,E1 18217.94,E2 18217.94} C_VEL
LIN {X 0,Y 444.461,Z 440.265,A -85,B 0,C 180,E1 18215.597,E2 18215.597} C_VEL
LIN {X 0,Y 432.913,Z 423.461,A -85,B 0,C 180,E1 18213.029,E2 18213.029} C_VEL
LIN {X 0,Y 424.421,Z 411.987,A -85,B 0,C 180,E1 18210.98,E2 18210.98} C_VEL
LIN {X 0,Y 416.984,Z 402.134,A -85,B 0,C 180,E1 18209.049,E2 18209.049} C_VEL
LIN {X 0,Y 413.412,Z 397.467,A -85,B 0,C 180,E1 18208.06,E2 18208.06} C_VEL
LIN {X 0,Y 410.008,Z 393.019,A -85,B 0,C 180,E1 18207.091,E2 18207.091} C_VEL
LIN {X 0,Y 405.714,Z 387.854,A -85,B 0,C 180,E1 18205.822,E2 18205.822} C_VEL
LIN {X 0,Y 404.349,Z 386.278,A -85,B 0,C 180,E1 18205.405,E2 18205.405} C_VEL
LIN {X 0,Y 402.014,Z 383.204,A -85,B 0,C 180,E1 18204.541,E2 18204.541} C_VEL
LIN {X 0,Y 401.49,Z 381.193,A -85,B 0,C 180,E1 18203.949,E2 18203.949} C_VEL
LIN {X 0,Y 401.45,Z 381.03,A -85,B 0,C 180,E1 18200.102,E2 18200.102} C_VEL
LIN {X 0,Y 401.435,Z 381.038,A -85,B 0,C 180,E1 18196.346,E2 18196.346} C_VEL
LIN {X 0,Y 401.435,Z 381.045,A -85,B 0,C 180,E1 18192.51,E2 18192.51} C_VEL
LIN {X 0,Y 401.439,Z 381.034,A -85,B 0,C 180,E1 18188.594,E2 18188.594} C_VEL
LIN {X 0,Y 401.461,Z 381.027,A -85,B 0,C 180,E1 18184.857,E2 18184.857} C_VEL
LIN {X 0,Y 401.486,Z 381.025,A -85,B 0,C 180,E1 18180.998,E2 18180.998} C_VEL
LIN {X 0,Y 401.486,Z 381.026,A -85,B 0,C 180,E1 18177.145,E2 18177.145} C_VEL
LIN {X 0,Y 401.475,Z 381.03,A -85,B 0,C 180,E1 18173.278,E2 18173.278} C_VEL
LIN {X 0,Y 401.464,Z 381.036,A -85,B 0,C 180,E1 18169.379,E2 18169.379} C_VEL
LIN {X 0,Y 401.455,Z 381.04,A -85,B 0,C 180,E1 18165.578,E2 18165.578} C_VEL
LIN {X 0,Y 401.46,Z 381.041,A -85,B 0,C 180,E1 18161.586,E2 18161.586} C_VEL
LIN {X 0,Y 401.461,Z 381.039,A -85,B 0,C 180,E1 18157.601,E2 18157.601} C_VEL
LIN {X 0,Y 401.47,Z 381.032,A -85,B 0,C 180,E1 18153.684,E2 18153.684} C_VEL
LIN {X 0,Y 401.498,Z 381.025,A -85,B 0,C 180,E1 18149.963,E2 18149.963} C_VEL
LIN {X 0,Y 401.502,Z 381.022,A -85,B 0,C 180,E1 18146.014,E2 18146.014} C_VEL
LIN {X 0,Y 401.506,Z 381.024,A -85,B 0,C 180,E1 18142.041,E2 18142.041} C_VEL
LIN {X 0,Y 401.504,Z 381.031,A -85,B 0,C 180,E1 18138.116,E2 18138.116} C_VEL
LIN {X 0,Y 401.495,Z 381.033,A -85,B 0,C 180,E1 18134.174,E2 18134.174} C_VEL
LIN {X 0,Y 401.486,Z 381.027,A -85,B 0,C 180,E1 18130.347,E2 18130.347} C_VEL
LIN {X 0,Y 401.481,Z 381.03,A -85,B 0,C 180,E1 18126.446,E2 18126.446} C_VEL
LIN {X 0,Y 401.526,Z 381.223,A -85,B 0,C 180,E1 18123.127,E2 18123.127} C_VEL
LIN {X 0,Y 401.854,Z 382.627,A -85,B 0,C 180,E1 18122.722,E2 18122.722} C_VEL
LIN {X 0,Y 403.674,Z 385.582,A -85,B 0,C 180,E1 18122.102,E2 18122.102} C_VEL
LIN {X 0,Y 406.661,Z 387.975,A -85,B 0,C 180,E1 18121.231,E2 18121.231} C_VEL
LIN {X 0,Y 409.042,Z 391.685,A -85,B 0,C 180,E1 18120.497,E2 18120.497} C_VEL
LIN {X 0,Y 411.672,Z 394.09,A -85,B 0,C 180,E1 18119.774,E2 18119.774} C_VEL
LIN {X 0,Y 414.535,Z 398.115,A -85,B 0,C 180,E1 18118.966,E2 18118.966} C_VEL
LIN {X 0,Y 416.806,Z 400.432,A -85,B 0,C 180,E1 18118.376,E2 18118.376} C_VEL
LIN {X 0,Y 420.316,Z 404.758,A -85,B 0,C 180,E1 18117.463,E2 18117.463} C_VEL
LIN {X 0,Y 426.389,Z 412.484,A -85,B 0,C 180,E1 18115.935,E2 18115.935} C_VEL
LIN {X 0,Y 434.73,Z 423.17,A -85,B 0,C 180,E1 18113.983,E2 18113.983} C_VEL
LIN {X 0,Y 445.796,Z 438.091,A -85,B 0,C 180,E1 18111.599,E2 18111.599} C_VEL
LIN {X 0,Y 455.725,Z 452.369,A -85,B 0,C 180,E1 18109.614,E2 18109.614} C_VEL
LIN {X 0,Y 449.416,Z 606.174,A -85,B 0,C 180,E1 18106.753,E2 18106.753} C_VEL
LIN {X 0,Y 448.46,Z 613.87,A -85,B 0,C 180,E1 18106.703,E2 18106.703} C_VEL
LIN {X 0,Y 443.42,Z 634.45,A -85,B 0,C 180,E1 18106.923,E2 18106.923} C_VEL
LIN {X 0,Y 442.652,Z 641.056,A -85,B 0,C 180,E1 18106.873,E2 18106.873} C_VEL
LIN {X 0,Y 439.49,Z 715.656,A -85,B 0,C 180,E1 18105.463,E2 18105.463} C_VEL
LIN {X 0,Y 437.528,Z 738.468,A -85,B 0,C 180,E1 18104.83,E2 18104.83} C_VEL
LIN {X 0,Y 435.074,Z 760.831,A -85,B 0,C 180,E1 18103.993,E2 18103.993} C_VEL
LIN {X 0,Y 432.282,Z 780.81,A -85,B 0,C 180,E1 18103.029,E2 18103.029} C_VEL
LIN {X 0,Y 428.864,Z 802.257,A -85,B 0,C 180,E1 18101.767,E2 18101.767} C_VEL
LIN {X 0,Y 425.227,Z 821.832,A -85,B 0,C 180,E1 18100.359,E2 18100.359} C_VEL
LIN {X 0,Y 421.207,Z 841.746,A -85,B 0,C 180,E1 18098.666,E2 18098.666} C_VEL
LIN {X 0,Y 417.168,Z 860.085,A -85,B 0,C 180,E1 18096.81,E2 18096.81} C_VEL
LIN {X 0,Y 412.735,Z 879.349,A -85,B 0,C 180,E1 18094.512,E2 18094.512} C_VEL
LIN {X 0,Y 408.862,Z 895.646,A -85,B 0,C 180,E1 18092.239,E2 18092.239} C_VEL
LIN {X 0,Y 405.154,Z 911.085,A -85,B 0,C 180,E1 18089.714,E2 18089.714} C_VEL
LIN {X 0,Y 401.818,Z 925.439,A -85,B 0,C 180,E1 18087.001,E2 18087.001} C_VEL
LIN {X 0,Y 398.901,Z 938.39,A -85,B 0,C 180,E1 18084.098,E2 18084.098} C_VEL
LIN {X 0,Y 396.494,Z 950.23,A -85,B 0,C 180,E1 18081.001,E2 18081.001} C_VEL
LIN {X 0,Y 394.702,Z 960.114,A -85,B 0,C 180,E1 18077.91,E2 18077.91} C_VEL
LIN {X 0,Y 393.335,Z 969.225,A -85,B 0,C 180,E1 18074.456,E2 18074.456} C_VEL
LIN {X 0,Y 392.561,Z 975.952,A -85,B 0,C 180,E1 18071.278,E2 18071.278} C_VEL
LIN {X 0,Y 392.14,Z 981.309,A -85,B 0,C 180,E1 18067.984,E2 18067.984} C_VEL
LIN {X 0,Y 391.963,Z 985.214,A -85,B 0,C 180,E1 18064.621,E2 18064.621} C_VEL
LIN {X 0,Y 391.925,Z 987.499,A -85,B 0,C 180,E1 18061.336,E2 18061.336} C_VEL
LIN {X 0,Y 391.909,Z 988.304,A -85,B 0,C 180,E1 18058.119,E2 18058.119} C_VEL
LIN {X 0,Y 391.92,Z 987.598,A -85,B 0,C 180,E1 18054.787,E2 18054.787} C_VEL
LIN {X 0,Y 391.956,Z 985.427,A -85,B 0,C 180,E1 18051.503,E2 18051.503} C_VEL
LIN {X 0,Y 392.129,Z 981.827,A -85,B 0,C 180,E1 18048.276,E2 18048.276} C_VEL
LIN {X 0,Y 392.518,Z 976.558,A -85,B 0,C 180,E1 18044.912,E2 18044.912} C_VEL
LIN {X 0,Y 393.244,Z 970.048,A -85,B 0,C 180,E1 18041.772,E2 18041.772} C_VEL
LIN {X 0,Y 394.507,Z 961.575,A -85,B 0,C 180,E1 18038.447,E2 18038.447} C_VEL
LIN {X 0,Y 396.183,Z 952.03,A -85,B 0,C 180,E1 18035.393,E2 18035.393} C_VEL
LIN {X 0,Y 398.664,Z 939.895,A -85,B 0,C 180,E1 18032.121,E2 18032.121} C_VEL
LIN {X 0,Y 401.404,Z 927.65,A -85,B 0,C 180,E1 18029.326,E2 18029.326} C_VEL
LIN {X 0,Y 404.85,Z 912.957,A -85,B 0,C 180,E1 18026.474,E2 18026.474} C_VEL
LIN {X 0,Y 408.611,Z 897.486,A -85,B 0,C 180,E1 18023.89,E2 18023.89} C_VEL
LIN {X 0,Y 412.416,Z 881.5,A -85,B 0,C 180,E1 18021.624,E2 18021.624} C_VEL
LIN {X 0,Y 416.662,Z 863.498,A -85,B 0,C 180,E1 18019.42,E2 18019.42} C_VEL
LIN {X 0,Y 420.766,Z 844.926,A -85,B 0,C 180,E1 18017.494,E2 18017.494} C_VEL
LIN {X 0,Y 425.026,Z 824.365,A -85,B 0,C 180,E1 18015.696,E2 18015.696} C_VEL
LIN {X 0,Y 428.553,Z 805.632,A -85,B 0,C 180,E1 18014.319,E2 18014.319} C_VEL
LIN {X 0,Y 432.074,Z 784.476,A -85,B 0,C 180,E1 18013.029,E2 18013.029} C_VEL
LIN {X 0,Y 434.788,Z 765.477,A -85,B 0,C 180,E1 18012.08,E2 18012.08} C_VEL
LIN {X 0,Y 437.533,Z 741.997,A -85,B 0,C 180,E1 18011.155,E2 18011.155} C_VEL
LIN {X 0,Y 439.365,Z 721.647,A -85,B 0,C 180,E1 18010.557,E2 18010.557} C_VEL
LIN {X 0,Y 441.058,Z 690.015,A -85,B 0,C 180,E1 18009.903,E2 18009.903} C_VEL
LIN {X 0,Y 449.977,Z 496.573,A -85,B 0,C 180,E1 18006.211,E2 18006.211} C_VEL
LIN {X 0,Y 451.918,Z 456.59,A -85,B 0,C 180,E1 18005.415,E2 18005.415} C_VEL
LIN {X 0,Y 443.171,Z 443.378,A -85,B 0,C 180,E1 18003.331,E2 18003.331} C_VEL
LIN {X 0,Y 435.965,Z 433.281,A -85,B 0,C 180,E1 18001.413,E2 18001.413} C_VEL
LIN {X 0,Y 432.073,Z 428.019,A -85,B 0,C 180,E1 18000.266,E2 18000.266} C_VEL
LIN {X 0,Y 429.325,Z 424.315,A -85,B 0,C 180,E1 17999.4,E2 17999.4} C_VEL
LIN {X 0,Y 425.746,Z 419.587,A -85,B 0,C 180,E1 17998.184,E2 17998.184} C_VEL
LIN {X 0,Y 422.349,Z 415.189,A -85,B 0,C 180,E1 17996.917,E2 17996.917} C_VEL
LIN {X 0,Y 418.198,Z 410.309,A -85,B 0,C 180,E1 17995.166,E2 17995.166} C_VEL
LIN {X 0,Y 417.118,Z 408.527,A -85,B 0,C 180,E1 17994.636,E2 17994.636} C_VEL
LIN {X 0,Y 413.991,Z 405.681,A -85,B 0,C 180,E1 17993.055,E2 17993.055} C_VEL
LIN {X 0,Y 412.132,Z 402.378,A -85,B 0,C 180,E1 17991.834,E2 17991.834} C_VEL
LIN {X 0,Y 408.463,Z 399.6,A -85,B 0,C 180,E1 17988.993,E2 17988.993} C_VEL
LIN {X 0,Y 406.904,Z 396.449,A -85,B 0,C 180,E1 17986.501,E2 17986.501} C_VEL
